KUKA KRL program: MyProgram_255().src

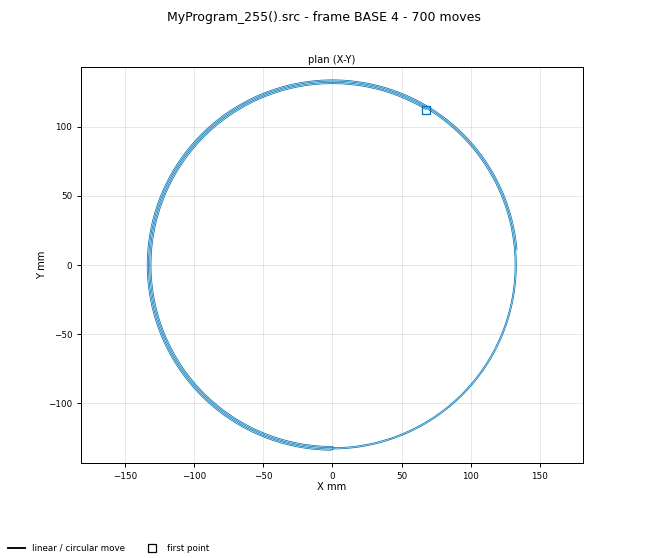
[picture p0: tool path of MyProgram_255().src in frame BASE 4, 700 of 700 moves have a stored position in this frame; points joined in program order, loops and branches not executed]
&ACCESS RVP
&REL 1
&PARAM TEMPLATE = C:\KRC\Roboter\Template\vorgabe
&PARAM EDITMASK = *
DEF MyProgram_255()
; ---- Setting reference (Base) ----
$BASE = BASE_DATA[4]

; --------------------------
; ---- Setting tool (TCP) ----
$TOOL = TOOL_DATA[3]
; --------------------------

$VEL.CP = VEL_APROX_PRINT
Startdeposition()
$VEL.CP = VEL_PRINT
LIN {X 67.662,Y 112.4887,Z 166,A 59.1873,B 11.341,C -0.0279,E1 11.4232,E2 391.3334} C_DIS
LIN {X 65.3064,Y 113.8724,Z 166,A 60.4715,B 11.341,C -0.0318,E1 11.4201,E2 390.0383} C_DIS
LIN {X 62.0567,Y 115.6751,Z 166,A 62.0322,B 11.341,C -0.0325,E1 11.4163,E2 388.4846} C_DIS
LIN {X 59.2043,Y 117.159,Z 166,A 63.3787,B 11.341,C -0.0329,E1 11.413,E2 387.1447} C_DIS
LIN {X 56.8476,Y 118.3202,Z 166,A 64.6326,B 11.341,C -0.037,E1 11.4098,E2 385.8781} C_DIS
LIN {X 53.382,Y 119.9236,Z 166,A 66.0531,B 11.341,C -0.0329,E1 11.4062,E2 384.4865} C_DIS
LIN {X 50.4227,Y 121.1975,Z 166,A 67.573,B 11.341,C -0.0372,E1 11.4023,E2 382.9533} C_DIS
LIN {X 47.4266,Y 122.401,Z 166,A 69.0048,B 11.341,C -0.0392,E1 11.3986,E2 381.519} C_DIS
LIN {X 44.4132,Y 123.5263,Z 166,A 70.3732,B 11.341,C -0.0397,E1 11.395,E2 380.1549} C_DIS
LIN {X 41.3721,Y 124.5778,Z 166,A 71.7718,B 11.341,C -0.0408,E1 11.3913,E2 378.7571} C_DIS
LIN {X 38.1151,Y 125.613,Z 166,A 73.257,B 11.341,C -0.0419,E1 11.3873,E2 377.2729} C_DIS
LIN {X 35.2196,Y 126.4551,Z 166,A 74.5585,B 11.341,C -0.0425,E1 11.3839,E2 375.9733} C_DIS
LIN {X 32.0679,Y 127.291,Z 166,A 75.9822,B 11.341,C -0.0435,E1 11.38,E2 374.5498} C_DIS
LIN {X 28.7806,Y 128.075,Z 166,A 77.4539,B 11.341,C -0.0443,E1 11.376,E2 373.0789} C_DIS
LIN {X 25.8073,Y 128.7068,Z 166,A 78.7946,B 11.341,C -0.0454,E1 11.3723,E2 371.7369} C_DIS
LIN {X 22.4469,Y 129.3365,Z 166,A 80.2607,B 11.341,C -0.0454,E1 11.3683,E2 370.2742} C_DIS
LIN {X 19.269,Y 129.8482,Z 166,A 81.6917,B 11.341,C -0.0466,E1 11.3644,E2 368.8407} C_DIS
LIN {X 16.0704,Y 130.2819,Z 166,A 83.0265,B 11.341,C -0.0453,E1 11.3607,E2 367.515} C_DIS
LIN {X 13.0675,Y 130.6173,Z 166,A 84.4622,B 11.341,C -0.0484,E1 11.3567,E2 366.0661} C_DIS
LIN {X 9.8613,Y 130.8977,Z 166,A 85.6593,B 11.341,C -0.0438,E1 11.3534,E2 364.8937} C_DIS
LIN {X 6.4486,Y 131.1099,Z 166,A 87.257,B 11.341,C -0.0464,E1 11.3489,E2 363.2843} C_DIS
LIN {X 3.2204,Y 131.2296,Z 166,A 88.6707,B 11.341,C -0.0466,E1 11.345,E2 361.8708} C_DIS
LIN {X 0.0025,Y 131.2704,Z 166,A 90.0792,B 11.341,C -0.0466,E1 11.341,E2 360.4626} C_DIS
LIN {X -3.2137,Y 131.2298,Z 166,A 91.4674,B 11.341,C -0.0461,E1 11.3372,E2 359.0768} C_DIS
LIN {X -6.4327,Y 131.1107,Z 166,A 92.8778,B 11.341,C -0.046,E1 11.3332,E2 357.6666} C_DIS
LIN {X -9.24,Y 130.9431,Z 166,A 94.2375,B 11.341,C -0.0487,E1 11.3294,E2 356.2921} C_DIS
LIN {X -12.6657,Y 130.6559,Z 166,A 95.6747,B 11.341,C -0.0468,E1 11.3254,E2 354.8631} C_DIS
LIN {X -16.0633,Y 130.2827,Z 166,A 97.1226,B 11.341,C -0.0452,E1 11.3214,E2 353.4212} C_DIS
LIN {X -19.0538,Y 129.8789,Z 166,A 98.4579,B 11.341,C -0.045,E1 11.3177,E2 352.0846} C_DIS
LIN {X -22.2446,Y 129.3713,Z 166,A 99.871,B 11.341,C -0.0443,E1 11.3138,E2 350.6721} C_DIS
LIN {X -25.4107,Y 128.7875,Z 166,A 101.3711,B 11.341,C -0.0456,E1 11.3097,E2 349.1619} C_DIS
LIN {X -28.5856,Y 128.1195,Z 166,A 102.7152,B 11.341,C -0.043,E1 11.306,E2 347.8271} C_DIS
LIN {X -31.9004,Y 127.3335,Z 166,A 104.1398,B 11.341,C -0.0405,E1 11.3022,E2 346.4108} C_DIS
LIN {X -34.8149,Y 126.5683,Z 166,A 105.5832,B 11.341,C -0.0423,E1 11.2983,E2 344.9533} C_DIS
LIN {X -37.9001,Y 125.6788,Z 166,A 106.9303,B 11.341,C -0.0398,E1 11.2947,E2 343.6137} C_DIS
LIN {X -41.1562,Y 124.6497,Z 166,A 108.4262,B 11.341,C -0.0385,E1 11.2907,E2 342.1182} C_DIS
LIN {X -44.2174,Y 123.5969,Z 166,A 109.8141,B 11.341,C -0.0365,E1 11.2871,E2 340.7344} C_DIS
LIN {X -47.0535,Y 122.546,Z 166,A 111.2316,B 11.341,C -0.0372,E1 11.2833,E2 339.3066} C_DIS
LIN {X -50.9887,Y 120.9611,Z 166,A 113.1889,B 11.341,C -0.0374,E1 11.2783,E2 337.3384} C_DIS
LIN {X -54.5865,Y 119.3812,Z 166,A 114.7862,B 11.341,C -0.0326,E1 11.2742,E2 335.7564} C_DIS
LIN {X -57.4016,Y 118.0545,Z 166,A 116.1867,B 11.341,C -0.0317,E1 11.2707,E2 334.3522} C_DIS
LIN {X -60.445,Y 116.5249,Z 166,A 117.565,B 11.341,C -0.0273,E1 11.2673,E2 332.9879} C_DIS
LIN {X -63.2703,Y 115.0164,Z 166,A 119.025,B 11.341,C -0.0266,E1 11.2637,E2 331.5219} C_DIS
LIN {X -66.0543,Y 113.4403,Z 166,A 120.4394,B 11.341,C -0.0249,E1 11.2603,E2 330.1066} C_DIS
LIN {X -68.7899,Y 111.8022,Z 166,A 121.854,B 11.341,C -0.0232,E1 11.2569,E2 328.6907} C_DIS
LIN {X -71.4124,Y 110.1455,Z 166,A 123.2027,B 11.341,C -0.0209,E1 11.2537,E2 327.3439} C_DIS
LIN {X -74.2646,Y 108.2429,Z 166,A 124.7098,B 11.341,C -0.0186,E1 11.2502,E2 325.837} C_DIS
LIN {X -76.7362,Y 106.5056,Z 166,A 126.0871,B 11.341,C -0.0175,E1 11.2471,E2 324.4541} C_DIS
LIN {X -79.4807,Y 104.4734,Z 166,A 127.6843,B 11.341,C -0.0171,E1 11.2435,E2 322.846} C_DIS
LIN {X -82.7236,Y 101.9251,Z 166,A 129.4945,B 11.341,C -0.0139,E1 11.2396,E2 321.0365} C_DIS
LIN {X -85.8192,Y 99.3321,Z 166,A 131.2791,B 11.341,C -0.0109,E1 11.2358,E2 319.2511} C_DIS
LIN {X -89.2655,Y 96.2471,Z 166,A 133.1947,B 11.341,C -0.0046,E1 11.2318,E2 317.3496} C_DIS
LIN {X -91.6701,Y 93.96,Z 166,A 134.657,B 11.341,C -0.0019,E1 11.2289,E2 315.8872} C_DIS
LIN {X -94.4472,Y 91.1675,Z 166,A 136.4062,B 11.341,C 0.0011,E1 11.2255,E2 314.1364} C_DIS
LIN {X -97.2631,Y 88.157,Z 166,A 138.3273,B 11.341,C 0.0026,E1 11.2218,E2 312.203} C_DIS
LIN {X -99.9831,Y 85.0597,Z 166,A 140.1409,B 11.341,C 0.0064,E1 11.2185,E2 310.3896} C_DIS
LIN {X -102.928,Y 81.4722,Z 166,A 142.0744,B 11.341,C 0.013,E1 11.2151,E2 308.4692} C_DIS
LIN {X -105.3163,Y 78.3596,Z 166,A 143.7874,B 11.341,C 0.0171,E1 11.2123,E2 306.758} C_DIS
LIN {X -107.3212,Y 75.5906,Z 166,A 145.2527,B 11.341,C 0.0212,E1 11.2099,E2 305.2975} C_DIS
LIN {X -109.0304,Y 73.104,Z 166,A 146.6964,B 11.341,C 0.0219,E1 11.2076,E2 303.8404} C_DIS
LIN {X -111.2462,Y 69.6864,Z 166,A 148.6229,B 11.341,C 0.0234,E1 11.2047,E2 301.8986} C_DIS
LIN {X -113.3192,Y 66.2616,Z 166,A 150.1978,B 11.341,C 0.0314,E1 11.2025,E2 300.3459} C_DIS
LIN {X -114.9075,Y 63.4669,Z 166,A 151.6157,B 11.341,C 0.0347,E1 11.2006,E2 298.9278} C_DIS
LIN {X -116.3051,Y 60.8637,Z 166,A 152.958,B 11.341,C 0.037,E1 11.1988,E2 297.5807} C_DIS
LIN {X -117.8767,Y 57.7619,Z 166,A 154.4808,B 11.341,C 0.041,E1 11.1969,E2 296.0591} C_DIS
LIN {X -119.2606,Y 54.8472,Z 166,A 155.8832,B 11.341,C 0.0449,E1 11.1952,E2 294.6589} C_DIS
LIN {X -120.5647,Y 51.9176,Z 166,A 157.2991,B 11.341,C 0.0483,E1 11.1937,E2 293.2427} C_DIS
LIN {X -121.7957,Y 48.9599,Z 166,A 158.7219,B 11.341,C 0.0517,E1 11.1922,E2 291.8187} C_DIS
LIN {X -123.0456,Y 45.7291,Z 166,A 160.2206,B 11.341,C 0.0562,E1 11.1907,E2 290.3232} C_DIS
LIN {X -124.0643,Y 42.8875,Z 166,A 161.581,B 11.341,C 0.059,E1 11.1894,E2 288.9594} C_DIS
LIN {X -125.0789,Y 39.8318,Z 166,A 163.141,B 11.3409,C 0.0598,E1 11.1881,E2 287.3828} C_DIS
LIN {X -126.4587,Y 35.2069,Z 166,A 165.1656,B 11.3409,C 0.0675,E1 11.1865,E2 285.3702} C_DIS
LIN {X -127.3329,Y 31.9028,Z 166,A 166.6254,B 11.3409,C 0.0724,E1 11.1855,E2 283.9159} C_DIS
LIN {X -128.0762,Y 28.7751,Z 166,A 167.9722,B 11.3408,C 0.0776,E1 11.1846,E2 282.5773} C_DIS
LIN {X -128.7073,Y 25.805,Z 166,A 169.4267,B 11.3408,C 0.0788,E1 11.1838,E2 281.1091} C_DIS
LIN {X -129.3345,Y 22.4582,Z 166,A 170.9103,B 11.3408,C 0.0832,E1 11.1831,E2 279.6275} C_DIS
LIN {X -129.8441,Y 19.2974,Z 166,A 172.3494,B 11.3408,C 0.0865,E1 11.1825,E2 278.185} C_DIS
LIN {X -130.2753,Y 16.1257,Z 166,A 173.682,B 11.3407,C 0.0919,E1 11.182,E2 276.8616} C_DIS
LIN {X -130.6063,Y 13.1817,Z 166,A 175.01,B 11.3407,C 0.0949,E1 11.1816,E2 275.5308} C_DIS
LIN {X -130.8983,Y 9.8531,Z 166,A 176.5923,B 11.3407,C 0.0967,E1 11.1812,E2 273.9355} C_DIS
LIN {X -131.1104,Y 6.4391,Z 166,A 177.9677,B 11.3406,C 0.1035,E1 11.181,E2 272.5755} C_DIS
LIN {X -131.2295,Y 3.2217,Z 166,A 179.447,B 11.3406,C 0.1061,E1 11.1809,E2 271.089} C_DIS
LIN {X -131.2723,Y 0.0074,Z 166,A -179.0626,B 11.3406,C 0.1085,E1 11.1809,E2 269.5899} C_DIS
LIN {X -131.1873,Y -4.6366,Z 166,A -176.9792,B 11.3405,C 0.1133,E1 11.181,E2 267.5019} C_DIS
LIN {X -131.0335,Y -7.8515,Z 166,A -175.6128,B 11.3405,C 0.1182,E1 11.1812,E2 266.1414} C_DIS
LIN {X -130.7845,Y -11.2613,Z 166,A -174.14,B 11.3404,C 0.123,E1 11.1815,E2 264.6724} C_DIS
LIN {X -130.4695,Y -14.4651,Z 166,A -172.7858,B 11.3404,C 0.1281,E1 11.1819,E2 263.3257} C_DIS
LIN {X -130.0967,Y -17.5042,Z 166,A -171.3374,B 11.3404,C 0.1297,E1 11.1824,E2 261.8653} C_DIS
LIN {X -129.6322,Y -20.6682,Z 166,A -169.9236,B 11.3403,C 0.1334,E1 11.183,E2 260.4508} C_DIS
LIN {X -129.0909,Y -23.8195,Z 166,A -168.5079,B 11.3403,C 0.137,E1 11.1837,E2 259.034} C_DIS
LIN {X -128.4298,Y -27.1555,Z 166,A -167.0467,B 11.3402,C 0.1417,E1 11.1845,E2 257.577} C_DIS
LIN {X -127.7642,Y -30.1336,Z 166,A -165.5785,B 11.3402,C 0.1428,E1 11.1855,E2 256.0938} C_DIS
LIN {X -126.9882,Y -33.2511,Z 166,A -164.222,B 11.3402,C 0.1477,E1 11.1864,E2 254.744} C_DIS
LIN {X -126.079,Y -36.5443,Z 166,A -162.78,B 11.34,C 0.1528,E1 11.1875,E2 253.309} C_DIS
LIN {X -125.199,Y -39.4556,Z 166,A -161.3122,B 11.34,C 0.1537,E1 11.1887,E2 251.8258} C_DIS
LIN {X -124.1294,Y -42.6997,Z 166,A -159.8592,B 11.34,C 0.1585,E1 11.19,E2 250.3785} C_DIS
LIN {X -123.0445,Y -45.732,Z 166,A -158.5033,B 11.3399,C 0.1634,E1 11.1913,E2 249.0297} C_DIS
LIN {X -121.8872,Y -48.7329,Z 166,A -157.0137,B 11.3399,C 0.1654,E1 11.1928,E2 247.531} C_DIS
LIN {X -120.3465,Y -52.4224,Z 166,A -155.212,B 11.3399,C 0.1689,E1 11.1948,E2 245.7239} C_DIS
LIN {X -118.6723,Y -56.1107,Z 166,A -153.5507,B 11.3397,C 0.1758,E1 11.1967,E2 244.0767} C_DIS
LIN {X -117.5193,Y -58.4864,Z 166,A -152.1926,B 11.3397,C 0.1745,E1 11.1984,E2 242.6951} C_DIS
LIN {X -115.6777,Y -62.0519,Z 166,A -150.4062,B 11.3397,C 0.1782,E1 11.2008,E2 240.9058} C_DIS
LIN {X -113.4207,Y -66.0882,Z 166,A -148.4733,B 11.3396,C 0.1851,E1 11.2034,E2 238.9844} C_DIS
LIN {X -111.7576,Y -68.8628,Z 166,A -147.0469,B 11.3396,C 0.1882,E1 11.2055,E2 237.5572} C_DIS
LIN {X -110.3098,Y -71.1593,Z 166,A -145.7766,B 11.3395,C 0.1893,E1 11.2074,E2 236.2774} C_DIS
LIN {X -108.241,Y -74.2674,Z 166,A -144.1303,B 11.3395,C 0.1928,E1 11.21,E2 234.6302} C_DIS
LIN {X -105.7565,Y -77.7645,Z 166,A -142.2177,B 11.3394,C 0.1963,E1 11.2131,E2 232.7138} C_DIS
LIN {X -103.4932,Y -80.7533,Z 166,A -140.5087,B 11.3394,C 0.1985,E1 11.2161,E2 230.9971} C_DIS
LIN {X -100.8567,Y -84.0229,Z 166,A -138.712,B 11.3393,C 0.2033,E1 11.2192,E2 229.2057} C_DIS
LIN {X -98.2956,Y -87.0043,Z 166,A -136.9297,B 11.3393,C 0.2055,E1 11.2225,E2 227.4161} C_DIS
LIN {X -95.6929,Y -89.8595,Z 166,A -135.327,B 11.3391,C 0.2108,E1 11.2256,E2 225.8243} C_DIS
LIN {X -92.8239,Y -92.8206,Z 166,A -133.4053,B 11.3391,C 0.2118,E1 11.2294,E2 223.8887} C_DIS
LIN {X -89.8627,Y -95.6898,Z 166,A -131.5943,B 11.3391,C 0.2151,E1 11.233,E2 222.0769} C_DIS
LIN {X -86.5059,Y -98.7347,Z 166,A -129.6375,B 11.339,C 0.2192,E1 11.2371,E2 220.1234} C_DIS
LIN {X -83.2718,Y -101.4773,Z 166,A -127.8857,B 11.3389,C 0.2247,E1 11.2408,E2 218.384} C_DIS
LIN {X -80.1684,Y -103.9465,Z 166,A -125.9969,B 11.3389,C 0.2242,E1 11.245,E2 216.4768} C_DIS
LIN {X -77.067,Y -106.2659,Z 166,A -124.4918,B 11.3387,C 0.2311,E1 11.2483,E2 214.9944} C_DIS
LIN {X -74.4424,Y -108.1209,Z 166,A -123.0232,B 11.3387,C 0.2318,E1 11.2517,E2 213.5181} C_DIS
LIN {X -72.1579,Y -109.6586,Z 166,A -121.6777,B 11.3387,C 0.2305,E1 11.2549,E2 212.1556} C_DIS
LIN {X -69.0408,Y -111.648,Z 166,A -120.1753,B 11.3387,C 0.2353,E1 11.2584,E2 210.6669} C_DIS
LIN {X -66.2691,Y -113.3148,Z 166,A -118.7593,B 11.3387,C 0.2372,E1 11.2618,E2 209.2505} C_DIS
LIN {X -63.9002,Y -114.6676,Z 166,A -117.4579,B 11.3387,C 0.2363,E1 11.265,E2 207.936} C_DIS
LIN {X -60.4624,Y -116.5158,Z 166,A -115.8994,B 11.3385,C 0.2417,E1 11.2688,E2 206.395} C_DIS
LIN {X -57.8004,Y -117.8577,Z 166,A -114.5216,B 11.3385,C 0.2415,E1 11.2723,E2 205.008} C_DIS
LIN {X -55.105,Y -119.1414,Z 166,A -113.1832,B 11.3385,C 0.2422,E1 11.2757,E2 203.6653} C_DIS
LIN {X -51.907,Y -120.5693,Z 166,A -111.6942,B 11.3385,C 0.2447,E1 11.2795,E2 202.1811} C_DIS
LIN {X -48.9276,Y -121.8087,Z 166,A -110.2816,B 11.3385,C 0.246,E1 11.2831,E2 200.7679} C_DIS
LIN {X -45.7401,Y -123.0415,Z 166,A -108.8104,B 11.3384,C 0.2479,E1 11.287,E2 199.2991} C_DIS
LIN {X -42.898,Y -124.0607,Z 166,A -107.4616,B 11.3384,C 0.2483,E1 11.2905,E2 197.9464} C_DIS
LIN {X -39.8469,Y -125.074,Z 166,A -106.0229,B 11.3384,C 0.2486,E1 11.2944,E2 196.5033} C_DIS
LIN {X -36.6683,Y -126.0428,Z 166,A -104.616,B 11.3384,C 0.2506,E1 11.2981,E2 195.1014} C_DIS
LIN {X -33.4679,Y -126.9304,Z 166,A -103.1835,B 11.3383,C 0.252,E1 11.302,E2 193.6707} C_DIS
LIN {X -30.5578,Y -127.6619,Z 166,A -101.8046,B 11.3383,C 0.2511,E1 11.3058,E2 192.2832} C_DIS
LIN {X -27.1923,Y -128.4218,Z 166,A -100.3413,B 11.3383,C 0.2529,E1 11.3097,E2 190.8247} C_DIS
LIN {X -24.3174,Y -128.9965,Z 166,A -99.0195,B 11.3383,C 0.2524,E1 11.3134,E2 189.4974} C_DIS
LIN {X -21.2035,Y -129.545,Z 166,A -97.62,B 11.3383,C 0.2524,E1 11.3172,E2 188.0951} C_DIS
LIN {X -17.6666,Y -130.0754,Z 166,A -96.082,B 11.3383,C 0.2535,E1 11.3215,E2 186.5595} C_DIS
LIN {X -14.6746,Y -130.447,Z 166,A -94.7613,B 11.3383,C 0.2536,E1 11.3251,E2 185.2377} C_DIS
LIN {X -11.2704,Y -130.7838,Z 166,A -93.3281,B 11.3383,C 0.2552,E1 11.3291,E2 183.8112} C_DIS
LIN {X -7.3216,Y -131.066,Z 166,A -91.3755,B 11.3383,C 0.25,E1 11.3346,E2 181.8308} C_DIS
LIN {X -3.2255,Y -131.2294,Z 166,A -89.7976,B 11.3383,C 0.255,E1 11.339,E2 180.2776} C_DIS
LIN {X -0.0098,Y -131.2704,Z 166,A -88.3914,B 11.3383,C 0.2548,E1 11.3429,E2 178.8705} C_DIS
LIN {X -0.0098,Y -131.2704,Z 166,A -88.3914,B 11.3383,C 0.2548,E1 11.3429,E2 178.8705} C_DIS
Enddeposition()
LIN {X 0.9627,Y -132.1793,Z 166,A -87.9974,B 11.3378,C 0.2622,E1 11.3437,E2 178.5145} C_DIS
Startdeposition()
$VEL.CP = VEL_PRINT
LIN {X -3.5481,Y -132.1372,Z 166,A -90.5843,B 11.3375,C 0.2775,E1 11.3362,E2 181.179} C_DIS
LIN {X -6.8903,Y -132.0053,Z 166,A -91.9427,B 11.3375,C 0.2753,E1 11.3325,E2 182.5269} C_DIS
LIN {X -10.7823,Y -131.7447,Z 166,A -93.783,B 11.3375,C 0.2787,E1 11.3273,E2 184.386} C_DIS
LIN {X -14.7745,Y -131.3579,Z 166,A -95.3648,B 11.3375,C 0.2747,E1 11.3229,E2 185.9496} C_DIS
LIN {X -17.6438,Y -131.0027,Z 166,A -96.5893,B 11.3375,C 0.2737,E1 11.3195,E2 187.171} C_DIS
LIN {X -20.5621,Y -130.576,Z 166,A -98.0041,B 11.3375,C 0.2765,E1 11.3156,E2 188.6027} C_DIS
LIN {X -25.0988,Y -129.7801,Z 166,A -100.0228,B 11.3375,C 0.2762,E1 11.31,E2 190.6245} C_DIS
LIN {X -28.9268,Y -128.9816,Z 166,A -101.6475,B 11.3375,C 0.2738,E1 11.3056,E2 192.2413} C_DIS
LIN {X -34.998,Y -127.4687,Z 166,A -104.2527,B 11.3376,C 0.2697,E1 11.2986,E2 194.8342} C_DIS
LIN {X -40.1602,Y -125.936,Z 166,A -106.718,B 11.3376,C 0.271,E1 11.292,E2 197.3157} C_DIS
LIN {X -43.9608,Y -124.6621,Z 166,A -108.3852,B 11.3376,C 0.268,E1 11.2876,E2 198.9747} C_DIS
LIN {X -48.0714,Y -123.1335,Z 166,A -110.3817,B 11.3376,C 0.2684,E1 11.2824,E2 200.9827} C_DIS
LIN {X -51.2743,Y -121.835,Z 166,A -111.8429,B 11.3377,C 0.266,E1 11.2786,E2 202.4396} C_DIS
LIN {X -55.0333,Y -120.1842,Z 166,A -113.6609,B 11.3377,C 0.265,E1 11.2739,E2 204.2621} C_DIS
LIN {X -59.3109,Y -118.1331,Z 166,A -115.6519,B 11.3378,C 0.2611,E1 11.269,E2 206.2454} C_DIS
LIN {X -62.9156,Y -116.254,Z 166,A -117.5195,B 11.3378,C 0.2612,E1 11.2643,E2 208.1255} C_DIS
LIN {X -66.402,Y -114.2979,Z 166,A -119.2831,B 11.3378,C 0.2596,E1 11.26,E2 209.8926} C_DIS
LIN {X -69.7189,Y -112.3054,Z 166,A -120.8703,B 11.338,C 0.2552,E1 11.2563,E2 211.4688} C_DIS
LIN {X -72.6717,Y -110.4175,Z 166,A -122.5068,B 11.338,C 0.2555,E1 11.2524,E2 213.1191} C_DIS
LIN {X -76.4072,Y -107.8666,Z 166,A -124.3738,B 11.338,C 0.2504,E1 11.2482,E2 214.9745} C_DIS
LIN {X -79.3283,Y -105.7372,Z 166,A -125.9122,B 11.3382,C 0.2472,E1 11.2447,E2 216.5091} C_DIS
LIN {X -81.708,Y -103.9086,Z 166,A -127.3283,B 11.3382,C 0.2475,E1 11.2416,E2 217.9386} C_DIS
LIN {X -86.5739,Y -99.8906,Z 166,A -130.0328,B 11.3382,C 0.2419,E1 11.2358,E2 220.6387} C_DIS
LIN {X -89.4536,Y -97.3204,Z 166,A -131.8115,B 11.3382,C 0.241,E1 11.2321,E2 222.4293} C_DIS
LIN {X -92.6327,Y -94.2994,Z 166,A -133.7286,B 11.3384,C 0.2376,E1 11.2282,E2 224.3476} C_DIS
LIN {X -95.7987,Y -91.082,Z 166,A -135.7454,B 11.3384,C 0.235,E1 11.2243,E2 226.3708} C_DIS
LIN {X -100.2187,Y -86.1938,Z 166,A -138.4156,B 11.3386,C 0.225,E1 11.2194,E2 229.0175} C_DIS
LIN {X -102.9955,Y -82.8561,Z 166,A -140.4726,B 11.3386,C 0.2245,E1 11.2157,E2 231.0944} C_DIS
LIN {X -105.3656,Y -79.8207,Z 166,A -142.1033,B 11.3387,C 0.2199,E1 11.2129,E2 232.7196} C_DIS
LIN {X -107.296,Y -77.2069,Z 166,A -143.6343,B 11.3387,C 0.2193,E1 11.2104,E2 234.2643} C_DIS
LIN {X -109.424,Y -74.1592,Z 166,A -145.2603,B 11.3387,C 0.2158,E1 11.2078,E2 235.8912} C_DIS
LIN {X -111.7157,Y -70.6599,Z 166,A -146.9595,B 11.3389,C 0.209,E1 11.2052,E2 237.5757} C_DIS
LIN {X -113.759,Y -67.3221,Z 166,A -148.8423,B 11.3389,C 0.2087,E1 11.2025,E2 239.4796} C_DIS
LIN {X -115.549,Y -64.2002,Z 166,A -150.2105,B 11.3391,C 0.2008,E1 11.2007,E2 240.824} C_DIS
LIN {X -117.4167,Y -60.7179,Z 166,A -152.0082,B 11.3391,C 0.1982,E1 11.1983,E2 242.6305} C_DIS
LIN {X -120.4535,Y -54.4416,Z 166,A -155.1893,B 11.3391,C 0.1936,E1 11.1945,E2 245.8282} C_DIS
LIN {X -121.9218,Y -51.0664,Z 166,A -156.7285,B 11.3393,C 0.1882,E1 11.1928,E2 247.3595} C_DIS
LIN {X -123.2326,Y -47.8165,Z 166,A -158.3019,B 11.3393,C 0.1852,E1 11.1912,E2 248.9381} C_DIS
LIN {X -124.4563,Y -44.5356,Z 166,A -159.7167,B 11.3394,C 0.179,E1 11.1898,E2 250.3395} C_DIS
LIN {X -125.4508,Y -41.6512,Z 166,A -161.1009,B 11.3394,C 0.1766,E1 11.1886,E2 251.7298} C_DIS
LIN {X -126.49,Y -38.381,Z 166,A -162.936,B 11.3394,C 0.1795,E1 11.187,E2 253.6047} C_DIS
LIN {X -127.439,Y -35.1039,Z 166,A -164.1022,B 11.3396,C 0.169,E1 11.1862,E2 254.7328} C_DIS
LIN {X -128.2028,Y -32.2005,Z 166,A -165.441,B 11.3396,C 0.1661,E1 11.1853,E2 256.0748} C_DIS
LIN {X -129.1394,Y -28.211,Z 166,A -167.9125,B 11.3395,C 0.175,E1 11.1837,E2 258.6261} C_DIS
LIN {X -130.1453,Y -23.1299,Z 166,A -169.4206,B 11.3398,C 0.1538,E1 11.183,E2 260.0458} C_DIS
LIN {X -131.0761,Y -17.0832,Z 166,A -172.1888,B 11.3398,C 0.1485,E1 11.1819,E2 262.8252} C_DIS
LIN {X -131.5276,Y -13.1748,Z 166,A -173.9683,B 11.3398,C 0.145,E1 11.1813,E2 264.6119} C_DIS
LIN {X -131.8436,Y -9.491,Z 166,A -175.6102,B 11.3399,C 0.1411,E1 11.181,E2 266.2567} C_DIS
LIN {X -132.0725,Y -5.4547,Z 166,A -177.3516,B 11.34,C 0.1357,E1 11.1807,E2 267.995} C_DIS
LIN {X -132.1683,Y -2.0896,Z 166,A -178.7968,B 11.34,C 0.1312,E1 11.1807,E2 269.4371} C_DIS
LIN {X -132.179,Y 1.437,Z 166,A 179.6148,B 11.3401,C 0.1279,E1 11.1807,E2 271.0309} C_DIS
LIN {X -132.0879,Y 5.0617,Z 166,A 178.0274,B 11.3401,C 0.1236,E1 11.1807,E2 272.6185} C_DIS
LIN {X -131.8611,Y 9.2516,Z 166,A 176.1759,B 11.3401,C 0.1189,E1 11.1811,E2 274.4719} C_DIS
LIN {X -131.5553,Y 12.8864,Z 166,A 174.6147,B 11.3403,C 0.1138,E1 11.1815,E2 276.029} C_DIS
LIN {X -130.7873,Y 19.1749,Z 166,A 171.5775,B 11.3403,C 0.1116,E1 11.1826,E2 279.0973} C_DIS
LIN {X -130.0788,Y 23.5011,Z 166,A 169.9122,B 11.3403,C 0.1014,E1 11.1834,E2 280.733} C_DIS
LIN {X -129.4416,Y 26.7919,Z 166,A 168.0038,B 11.3403,C 0.1063,E1 11.1845,E2 282.693} C_DIS
LIN {X -128.6,Y 30.5768,Z 166,A 166.6692,B 11.3404,C 0.0945,E1 11.1853,E2 283.9854} C_DIS
LIN {X -127.7264,Y 34.0396,Z 166,A 165.1741,B 11.3404,C 0.089,E1 11.1863,E2 285.4725} C_DIS
LIN {X -126.6616,Y 37.816,Z 166,A 163.4553,B 11.3405,C 0.0846,E1 11.1877,E2 287.1916} C_DIS
LIN {X -125.808,Y 40.561,Z 166,A 162.1921,B 11.3405,C 0.0814,E1 11.1887,E2 288.4554} C_DIS
LIN {X -124.8755,Y 43.3452,Z 166,A 160.8136,B 11.3405,C 0.0799,E1 11.19,E2 289.8448} C_DIS
LIN {X -123.7018,Y 46.5898,Z 166,A 159.3856,B 11.3405,C 0.0744,E1 11.1914,E2 291.2632} C_DIS
LIN {X -122.4123,Y 49.8815,Z 166,A 157.3407,B 11.3405,C 0.0804,E1 11.1936,E2 293.366} C_DIS
LIN {X -120.8023,Y 53.6618,Z 166,A 155.9611,B 11.3406,C 0.0676,E1 11.1951,E2 294.6969} C_DIS
LIN {X -118.8847,Y 57.7887,Z 166,A 154.0809,B 11.3406,C 0.0604,E1 11.1973,E2 296.5641} C_DIS
LIN {X -117.7882,Y 59.9884,Z 166,A 152.857,B 11.3406,C 0.0607,E1 11.1988,E2 297.8052} C_DIS
LIN {X -116.0492,Y 63.2912,Z 166,A 151.3783,B 11.3406,C 0.0537,E1 11.2008,E2 299.2659} C_DIS
LIN {X -114.2437,Y 66.4951,Z 166,A 149.7474,B 11.3407,C 0.0503,E1 11.203,E2 300.8994} C_DIS
LIN {X -111.878,Y 70.4027,Z 166,A 147.4577,B 11.3407,C 0.0516,E1 11.2064,E2 303.2228} C_DIS
LIN {X -109.2257,Y 74.4521,Z 166,A 145.444,B 11.3407,C 0.0447,E1 11.2095,E2 305.2244} C_DIS
LIN {X -106.7687,Y 77.9346,Z 166,A 143.566,B 11.3407,C 0.0408,E1 11.2126,E2 307.1039} C_DIS
LIN {X -104.2939,Y 81.2162,Z 166,A 141.7827,B 11.3407,C 0.0366,E1 11.2156,E2 308.8854} C_DIS
LIN {X -101.483,Y 84.7025,Z 166,A 139.8758,B 11.3407,C 0.0314,E1 11.219,E2 310.7862} C_DIS
LIN {X -98.7041,Y 87.9251,Z 166,A 138.036,B 11.3407,C 0.0271,E1 11.2224,E2 312.6235} C_DIS
LIN {X -95.9035,Y 90.9717,Z 166,A 136.2133,B 11.3407,C 0.0238,E1 11.2258,E2 314.4475} C_DIS
LIN {X -93.2084,Y 93.7304,Z 166,A 134.4678,B 11.3407,C 0.0218,E1 11.2293,E2 316.1998} C_DIS
LIN {X -90.1698,Y 96.6572,Z 166,A 132.6495,B 11.3408,C 0.0178,E1 11.233,E2 318.015} C_DIS
LIN {X -87.147,Y 99.3916,Z 166,A 130.8111,B 11.3408,C 0.0157,E1 11.2368,E2 319.8599} C_DIS
LIN {X -83.671,Y 102.3345,Z 166,A 128.852,B 11.3408,C 0.0116,E1 11.241,E2 321.8152} C_DIS
LIN {X -80.4137,Y 104.9135,Z 166,A 127.0637,B 11.3408,C 0.008,E1 11.2449,E2 323.6003} C_DIS
LIN {X -77.3577,Y 107.187,Z 166,A 125.3784,B 11.3408,C 0.0058,E1 11.2487,E2 325.2879} C_DIS
LIN {X -73.6429,Y 109.7726,Z 166,A 123.3812,B 11.3408,C 0.0032,E1 11.2534,E2 327.2873} C_DIS
LIN {X -69.84,Y 112.23,Z 166,A 121.4918,B 11.3408,C -0.0016,E1 11.2578,E2 329.1664} C_DIS
LIN {X -64.4414,Y 115.4151,Z 166,A 118.6279,B 11.3408,C -0.0026,E1 11.2647,E2 332.0448} C_DIS
LIN {X -61.1977,Y 117.1648,Z 166,A 117.1535,B 11.3408,C -0.0075,E1 11.2683,E2 333.5035} C_DIS
LIN {X -58.2534,Y 118.6561,Z 166,A 115.724,B 11.3408,C -0.0095,E1 11.2719,E2 334.9315} C_DIS
LIN {X -52.6518,Y 121.2457,Z 166,A 112.9525,B 11.3408,C -0.0108,E1 11.279,E2 337.712} C_DIS
LIN {X -48.9305,Y 122.7956,Z 166,A 111.2223,B 11.3408,C -0.0132,E1 11.2834,E2 339.4388} C_DIS
LIN {X -44.7986,Y 124.3615,Z 166,A 109.2791,B 11.3408,C -0.0146,E1 11.2885,E2 341.3837} C_DIS
LIN {X -38.9801,Y 126.3066,Z 166,A 106.8985,B 11.3408,C -0.0233,E1 11.2948,E2 343.7299} C_DIS
LIN {X -34.8285,Y 127.516,Z 166,A 104.694,B 11.3408,C -0.0176,E1 11.3008,E2 345.9716} C_DIS
LIN {X -31.0574,Y 128.4842,Z 166,A 103.161,B 11.3408,C -0.0223,E1 11.3049,E2 347.4854} C_DIS
LIN {X -25.7992,Y 129.6436,Z 166,A 100.7895,B 11.3408,C -0.023,E1 11.3114,E2 349.8597} C_DIS
LIN {X -21.9761,Y 130.3452,Z 166,A 99.0916,B 11.3408,C -0.0237,E1 11.316,E2 351.558} C_DIS
LIN {X -18.6805,Y 130.858,Z 166,A 97.6643,B 11.3408,C -0.0248,E1 11.32,E2 352.9823} C_DIS
LIN {X -15.4361,Y 131.2804,Z 166,A 96.1226,B 11.3408,C -0.0226,E1 11.3243,E2 354.5375} C_DIS
LIN {X -10.9024,Y 131.7345,Z 166,A 94.1987,B 11.3408,C -0.0244,E1 11.3296,E2 356.4544} C_DIS
LIN {X -7.1231,Y 131.9936,Z 166,A 92.5139,B 11.3408,C -0.0238,E1 11.3343,E2 358.1434} C_DIS
LIN {X -3.5616,Y 132.1369,Z 166,A 90.9488,B 11.3408,C -0.0236,E1 11.3387,E2 359.7099} C_DIS
LIN {X 0.1908,Y 132.1858,Z 166,A 89.3327,B 11.3408,C -0.024,E1 11.3432,E2 361.3242} C_DIS
LIN {X 3.9208,Y 132.1269,Z 166,A 87.8581,B 11.3408,C -0.0272,E1 11.3473,E2 362.7814} C_DIS
LIN {X 7.3388,Y 131.9826,Z 166,A 86.3652,B 11.3408,C -0.0268,E1 11.3514,E2 364.275} C_DIS
LIN {X 11.482,Y 131.6856,Z 166,A 84.5479,B 11.3408,C -0.0261,E1 11.3565,E2 366.0934} C_DIS
LIN {X 14.2529,Y 131.414,Z 166,A 83.352,B 11.3408,C -0.0261,E1 11.3598,E2 367.2877} C_DIS
LIN {X 17.3054,Y 131.047,Z 166,A 81.9399,B 11.3408,C -0.0238,E1 11.3637,E2 368.7085} C_DIS
LIN {X 21.6847,Y 130.3938,Z 166,A 79.9789,B 11.3408,C -0.0221,E1 11.3692,E2 370.6739} C_DIS
LIN {X 25.7769,Y 129.6482,Z 166,A 78.1988,B 11.3408,C -0.0217,E1 11.374,E2 372.4509} C_DIS
LIN {X 31.3948,Y 128.4028,Z 166,A 75.7743,B 11.3408,C -0.0218,E1 11.3806,E2 374.8667} C_DIS
LIN {X 37.3211,Y 126.8065,Z 166,A 73.0355,B 11.3408,C -0.018,E1 11.388,E2 377.6142} C_DIS
LIN {X 40.7946,Y 125.7333,Z 166,A 71.5528,B 11.3408,C -0.0189,E1 11.3919,E2 379.0859} C_DIS
LIN {X 44.6681,Y 124.4086,Z 166,A 69.718,B 11.3408,C -0.0159,E1 11.3968,E2 380.9275} C_DIS
LIN {X 48.2829,Y 123.0513,Z 166,A 68.121,B 11.3408,C -0.016,E1 11.4009,E2 382.5155} C_DIS
LIN {X 52.1574,Y 121.4594,Z 166,A 66.3341,B 11.3408,C -0.0148,E1 11.4055,E2 384.299} C_DIS
LIN {X 55.5916,Y 119.9261,Z 166,A 64.6916,B 11.3408,C -0.0126,E1 11.4097,E2 385.9429} C_DIS
LIN {X 58.8648,Y 118.3545,Z 166,A 63.138,B 11.3408,C -0.0111,E1 11.4136,E2 387.4942} C_DIS
LIN {X 62.0016,Y 116.7427,Z 166,A 61.6458,B 11.3408,C -0.01,E1 11.4173,E2 388.9822} C_DIS
LIN {X 64.903,Y 115.1556,Z 166,A 60.0227,B 11.3408,C -0.0034,E1 11.4213,E2 390.6277} C_DIS
LIN {X 68.0801,Y 113.3069,Z 166,A 58.592,B 11.3408,C -0.005,E1 11.4247,E2 392.0397} C_DIS
LIN {X 71.4574,Y 111.2074,Z 166,A 56.7287,B 11.3408,C 0.001,E1 11.4291,E2 393.9196} C_DIS
LIN {X 75.1479,Y 108.7481,Z 166,A 54.8646,B 11.3408,C 0.0027,E1 11.4334,E2 395.7772} C_DIS
LIN {X 78.5579,Y 106.3108,Z 166,A 53.1359,B 11.3408,C 0.0035,E1 11.4373,E2 397.496} C_DIS
LIN {X 81.7351,Y 103.8873,Z 166,A 51.2943,B 11.3408,C 0.0093,E1 11.4414,E2 399.3509} C_DIS
LIN {X 84.2875,Y 101.8274,Z 166,A 49.9707,B 11.3408,C 0.0095,E1 11.4442,E2 400.6634} C_DIS
LIN {X 87.7168,Y 98.8888,Z 166,A 48.0574,B 11.3408,C 0.012,E1 11.4483,E2 402.5722} C_DIS
LIN {X 90.7514,Y 96.1113,Z 166,A 46.2601,B 11.3408,C 0.0159,E1 11.4519,E2 404.3718} C_DIS
LIN {X 93.6236,Y 93.3159,Z 166,A 44.5122,B 11.3408,C 0.0197,E1 11.4554,E2 406.1217} C_DIS
LIN {X 96.6964,Y 90.1277,Z 166,A 42.6164,B 11.3408,C 0.0231,E1 11.459,E2 408.0156} C_DIS
LIN {X 99.8334,Y 86.6407,Z 166,A 40.6337,B 11.3408,C 0.0262,E1 11.4627,E2 409.9933} C_DIS
LIN {X 103.3191,Y 82.4523,Z 166,A 38.2826,B 11.3408,C 0.0312,E1 11.4669,E2 412.3443} C_DIS
LIN {X 106.0108,Y 78.9614,Z 166,A 36.455,B 11.3408,C 0.0335,E1 11.4699,E2 414.1631} C_DIS
LIN {X 108.3485,Y 75.7223,Z 166,A 34.898,B 11.3408,C 0.033,E1 11.4724,E2 415.7005} C_DIS
LIN {X 109.7492,Y 73.6779,Z 166,A 33.7322,B 11.3408,C 0.038,E1 11.4743,E2 416.8778} C_DIS
LIN {X 111.5595,Y 70.9074,Z 166,A 32.1997,B 11.3408,C 0.044,E1 11.4766,E2 418.4228} C_DIS
LIN {X 114.3985,Y 66.2282,Z 166,A 30.107,B 11.3408,C 0.0427,E1 11.4796,E2 420.484} C_DIS
LIN {X 115.6749,Y 63.9728,Z 166,A 28.8023,B 11.3408,C 0.0502,E1 11.4814,E2 421.8109} C_DIS
LIN {X 117.4945,Y 60.5653,Z 166,A 26.9343,B 11.3407,C 0.0596,E1 11.4838,E2 423.703} C_DIS
LIN {X 119.592,Y 56.3115,Z 166,A 24.9848,B 11.3407,C 0.0622,E1 11.4862,E2 425.6415} C_DIS
LIN {X 121.3091,Y 52.5051,Z 166,A 23.3016,B 11.3407,C 0.0637,E1 11.4881,E2 427.3109} C_DIS
LIN {X 122.8718,Y 48.7417,Z 166,A 21.635,B 11.3407,C 0.0659,E1 11.4898,E2 428.9673} C_DIS
LIN {X 124.117,Y 45.4767,Z 166,A 20.1749,B 11.3407,C 0.0686,E1 11.4912,E2 430.4221} C_DIS
LIN {X 124.9594,Y 43.1034,Z 166,A 18.9844,B 11.3406,C 0.0741,E1 11.4923,E2 431.6251} C_DIS
LIN {X 126.0736,Y 39.7293,Z 166,A 17.4316,B 11.3406,C 0.0788,E1 11.4937,E2 433.1809} C_DIS
LIN {X 127.0794,Y 36.387,Z 166,A 15.9293,B 11.3406,C 0.0827,E1 11.4949,E2 434.6831} C_DIS
LIN {X 128.3596,Y 31.5742,Z 166,A 13.8012,B 11.3405,C 0.088,E1 11.4963,E2 436.8095} C_DIS
LIN {X 129.2165,Y 27.8538,Z 166,A 12.2557,B 11.3405,C 0.0899,E1 11.4973,E2 438.3436} C_DIS
LIN {X 129.9463,Y 24.2298,Z 166,A 10.6925,B 11.3405,C 0.0934,E1 11.4981,E2 439.9036} C_DIS
LIN {X 130.6123,Y 20.3276,Z 166,A 8.9698,B 11.3404,C 0.0986,E1 11.4989,E2 441.6287} C_DIS
LIN {X 131.106,Y 16.8548,Z 166,A 7.3603,B 11.3404,C 0.1054,E1 11.4995,E2 443.2503} C_DIS
LIN {X 131.5837,Y 12.5906,Z 166,A 5.6027,B 11.3404,C 0.1081,E1 11.5,E2 444.9976} C_DIS
LIN {X 131.9037,Y 8.6299,Z 166,A 3.8912,B 11.3403,C 0.1128,E1 11.5003,E2 446.7096} C_DIS
LIN {X 132.089,Y 5.0313,Z 166,A 2.4064,B 11.3403,C 0.1154,E1 11.5005,E2 448.1867} C_DIS
LIN {X 132.1809,Y 1.1603,Z 166,A 0.811,B 11.3403,C 0.1181,E1 11.5006,E2 449.7739} C_DIS
LIN {X 132.1666,Y -2.1972,Z 166,A -0.7243,B 11.3401,C 0.1245,E1 11.5006,E2 451.3203} C_DIS
LIN {X 132.0287,Y -6.4256,Z 166,A -2.5224,B 11.3401,C 0.129,E1 11.5004,E2 453.1161} C_DIS
LIN {X 131.803,Y -10.0466,Z 166,A -4.0423,B 11.3401,C 0.1322,E1 11.5001,E2 454.6314} C_DIS
LIN {X 131.5353,Y -13.0944,Z 166,A -5.3126,B 11.3401,C 0.1346,E1 11.4998,E2 455.8964} C_DIS
LIN {X 131.2109,Y -16.0188,Z 166,A -6.6099,B 11.34,C 0.139,E1 11.4993,E2 457.1977} C_DIS
LIN {X 130.6667,Y -19.976,Z 166,A -8.3004,B 11.34,C 0.1429,E1 11.4987,E2 458.8853} C_DIS
LIN {X 130.083,Y -23.4777,Z 166,A -9.8787,B 11.3399,C 0.1485,E1 11.4979,E2 460.4699} C_DIS
LIN {X 129.3554,Y -27.2107,Z 166,A -12.109,B 11.3396,C 0.1687,E1 11.4966,E2 462.7716} C_DIS
LIN {X 128.2416,Y -32.0478,Z 166,A -13.4592,B 11.3398,C 0.1537,E1 11.4958,E2 464.0285} C_DIS
LIN {X 127.0755,Y -36.4023,Z 166,A -15.5121,B 11.3397,C 0.1619,E1 11.4943,E2 466.0956} C_DIS
LIN {X 126.0127,Y -39.9201,Z 166,A -17.2474,B 11.3396,C 0.1702,E1 11.4928,E2 467.8497} C_DIS
LIN {X 124.8057,Y -43.5466,Z 166,A -18.8197,B 11.3396,C 0.1727,E1 11.4914,E2 469.4138} C_DIS
LIN {X 123.1785,Y -47.9557,Z 166,A -20.7476,B 11.3395,C 0.1755,E1 11.4895,E2 471.3309} C_DIS
LIN {X 121.8948,Y -51.1311,Z 166,A -22.2646,B 11.3394,C 0.1804,E1 11.4879,E2 472.8535} C_DIS
LIN {X 120.3524,Y -54.6678,Z 166,A -25.1269,B 11.3388,C 0.2162,E1 11.4844,E2 475.8594} C_DIS
LIN {X 116.6915,Y -62.0991,Z 166,A -27.9035,B 11.339,C 0.2045,E1 11.4809,E2 478.5437} C_DIS
LIN {X 114.6093,Y -65.8641,Z 166,A -29.2529,B 11.3391,C 0.1959,E1 11.4791,E2 479.8335} C_DIS
LIN {X 112.5775,Y -69.2786,Z 166,A -30.918,B 11.3391,C 0.1988,E1 11.4767,E2 481.4936} C_DIS
LIN {X 110.8795,Y -71.9648,Z 166,A -32.4089,B 11.339,C 0.2053,E1 11.4745,E2 482.9998} C_DIS
LIN {X 108.3155,Y -75.7697,Z 166,A -34.4093,B 11.3389,C 0.2106,E1 11.4713,E2 485.0037} C_DIS
LIN {X 105.7174,Y -79.3545,Z 166,A -36.3143,B 11.3389,C 0.2149,E1 11.4681,E2 486.9092} C_DIS
LIN {X 102.8405,Y -83.0483,Z 166,A -38.4527,B 11.3387,C 0.2226,E1 11.4644,E2 489.063} C_DIS
LIN {X 100.4393,Y -85.9379,Z 166,A -39.9266,B 11.3387,C 0.2223,E1 11.4618,E2 490.5202} C_DIS
LIN {X 97.4774,Y -89.2827,Z 166,A -41.7418,B 11.3387,C 0.2236,E1 11.4584,E2 492.3229} C_DIS
LIN {X 94.9714,Y -91.9436,Z 166,A -43.4125,B 11.3385,C 0.2293,E1 11.4552,E2 494.0057} C_DIS
LIN {X 91.7664,Y -95.143,Z 166,A -45.3124,B 11.3385,C 0.2319,E1 11.4514,E2 495.9001} C_DIS
LIN {X 88.973,Y -97.7601,Z 166,A -46.9798,B 11.3384,C 0.2356,E1 11.448,E2 497.5703} C_DIS
LIN {X 85.5432,Y -100.7748,Z 166,A -48.9725,B 11.3384,C 0.2399,E1 11.4437,E2 499.5666} C_DIS
LIN {X 82.54,Y -103.2493,Z 166,A -50.5289,B 11.3384,C 0.2399,E1 11.4404,E2 501.109} C_DIS
LIN {X 79.6998,Y -105.4568,Z 166,A -52.0576,B 11.3383,C 0.242,E1 11.437,E2 502.6356} C_DIS
LIN {X 77.2018,Y -107.2997,Z 166,A -53.5225,B 11.3381,C 0.2476,E1 11.4337,E2 504.1164} C_DIS
LIN {X 73.5506,Y -109.8341,Z 166,A -55.5192,B 11.3381,C 0.2527,E1 11.429,E2 506.1234} C_DIS
LIN {X 69.9632,Y -112.1533,Z 166,A -57.2313,B 11.3381,C 0.2523,E1 11.425,E2 507.8204} C_DIS
LIN {X 66.5872,Y -114.1907,Z 166,A -58.8909,B 11.3381,C 0.2538,E1 11.4211,E2 509.4758} C_DIS
LIN {X 63.0428,Y -116.1847,Z 166,A -60.7469,B 11.3379,C 0.2589,E1 11.4165,E2 511.3446} C_DIS
LIN {X 59.3762,Y -118.0998,Z 166,A -62.3554,B 11.3379,C 0.2568,E1 11.4125,E2 512.9324} C_DIS
LIN {X 56.7675,Y -119.3741,Z 166,A -63.6195,B 11.3379,C 0.2587,E1 11.4094,E2 514.1983} C_DIS
LIN {X 53.9477,Y -120.6744,Z 166,A -64.9793,B 11.3379,C 0.2609,E1 11.4059,E2 515.5609} C_DIS
LIN {X 50.4453,Y -122.1812,Z 166,A -66.5654,B 11.3379,C 0.2613,E1 11.4018,E2 517.1405} C_DIS
LIN {X 47.0458,Y -123.531,Z 166,A -68.1303,B 11.3379,C 0.2627,E1 11.3978,E2 518.7042} C_DIS
LIN {X 44.1282,Y -124.6032,Z 166,A -69.8337,B 11.3376,C 0.273,E1 11.3932,E2 520.4516} C_DIS
LIN {X 40.9548,Y -125.6822,Z 166,A -70.9324,B 11.3377,C 0.2658,E1 11.3904,E2 521.5087} C_DIS
LIN {X 33.0839,Y -127.9786,Z 166,A -74.4959,B 11.3377,C 0.2694,E1 11.3808,E2 525.0761} C_DIS
LIN {X 30.2855,Y -128.6702,Z 166,A -75.9245,B 11.3375,C 0.2748,E1 11.3768,E2 526.5273} C_DIS
LIN {X 26.4865,Y -129.5038,Z 166,A -77.4272,B 11.3376,C 0.2715,E1 11.3728,E2 528.0089} C_DIS
LIN {X 22.6499,Y -130.2312,Z 166,A -79.0815,B 11.3376,C 0.2717,E1 11.3683,E2 529.6598} C_DIS
LIN {X 19.9028,Y -130.678,Z 166,A -80.3069,B 11.3376,C 0.2729,E1 11.3649,E2 530.8882} C_DIS
LIN {X 15.9178,Y -131.223,Z 166,A -82.1081,B 11.3376,C 0.2752,E1 11.3599,E2 532.6975} C_DIS
LIN {X 12.2971,Y -131.6119,Z 166,A -83.5528,B 11.3376,C 0.2726,E1 11.3559,E2 534.1269} C_DIS
LIN {X 8.9457,Y -131.8834,Z 166,A -85.2392,B 11.3374,C 0.2787,E1 11.3511,E2 535.8418} C_DIS
LIN {X 4.7739,Y -132.0991,Z 166,A -87.0037,B 11.3374,C 0.278,E1 11.3462,E2 537.6017} C_DIS
LIN {X 0.9627,Y -132.1793,Z 166,A -87.9958,B 11.3378,C 0.2625,E1 11.3437,E2 538.5145} C_DIS
Enddeposition()
LIN {X 0.9627,Y -132.1793,Z 166,A -87.9958,B 11.3378,C 0.2625,E1 11.3437,E2 538.5145} C_DIS
Startdeposition()
$VEL.CP = VEL_PRINT
LIN {X 1.6006,Y -133.093,Z 166,A -87.4623,B 11.3376,C 0.263,E1 11.345,E2 537.9838} C_DIS
LIN {X 5.8752,Y -132.9732,Z 166,A -85.6166,B 11.3376,C 0.2625,E1 11.3501,E2 536.1366} C_DIS
LIN {X 9.6604,Y -132.7501,Z 166,A -84.0983,B 11.3376,C 0.2647,E1 11.3543,E2 534.6314} C_DIS
LIN {X 13.7545,Y -132.3894,Z 166,A -82.3127,B 11.3376,C 0.2636,E1 11.3593,E2 532.8428} C_DIS
LIN {X 17.335,Y -131.9674,Z 166,A -80.7829,B 11.3376,C 0.2634,E1 11.3635,E2 531.3147} C_DIS
LIN {X 21.1406,Y -131.4137,Z 166,A -78.9869,B 11.3377,C 0.2589,E1 11.3685,E2 529.5005} C_DIS
LIN {X 24.9411,Y -130.7433,Z 166,A -77.5016,B 11.3377,C 0.2622,E1 11.3725,E2 528.0357} C_DIS
LIN {X 27.8456,Y -130.1558,Z 166,A -76.1901,B 11.3377,C 0.2604,E1 11.3761,E2 526.7189} C_DIS
LIN {X 32.0496,Y -129.1866,Z 166,A -73.6619,B 11.3381,C 0.2419,E1 11.3832,E2 524.1061} C_DIS
LIN {X 37.2295,Y -127.7882,Z 166,A -72.0253,B 11.3378,C 0.2568,E1 11.3874,E2 522.5514} C_DIS
LIN {X 44.175,Y -125.5578,Z 166,A -68.9626,B 11.3378,C 0.2555,E1 11.3955,E2 519.496} C_DIS
LIN {X 47.4817,Y -124.346,Z 166,A -67.4441,B 11.3378,C 0.2537,E1 11.3995,E2 517.9759} C_DIS
LIN {X 50.4857,Y -123.1568,Z 166,A -65.9525,B 11.3379,C 0.2494,E1 11.4034,E2 516.4708} C_DIS
LIN {X 54.1533,Y -121.5864,Z 166,A -64.3267,B 11.3379,C 0.2495,E1 11.4075,E2 514.8547} C_DIS
LIN {X 57.2062,Y -120.1802,Z 166,A -62.9342,B 11.3379,C 0.2489,E1 11.411,E2 513.4676} C_DIS
LIN {X 60.0301,Y -118.7953,Z 166,A -61.5284,B 11.338,C 0.2457,E1 11.4145,E2 512.0542} C_DIS
LIN {X 63.0442,Y -117.2252,Z 166,A -60.0441,B 11.338,C 0.2429,E1 11.4182,E2 510.566} C_DIS
LIN {X 66.9034,Y -115.0665,Z 166,A -58.1327,B 11.3381,C 0.2397,E1 11.4229,E2 508.6518} C_DIS
LIN {X 70.651,Y -112.8047,Z 166,A -55.7787,B 11.3384,C 0.2244,E1 11.4286,E2 506.2377} C_DIS
LIN {X 74.5977,Y -110.2338,Z 166,A -54.3149,B 11.3382,C 0.2356,E1 11.4318,E2 504.8419} C_DIS
LIN {X 77.7885,Y -108.0065,Z 166,A -52.5613,B 11.3383,C 0.2305,E1 11.4358,E2 503.077} C_DIS
LIN {X 81.2603,Y -105.4191,Z 166,A -50.6038,B 11.3384,C 0.2245,E1 11.4402,E2 501.106} C_DIS
LIN {X 86.5654,Y -101.1083,Z 166,A -47.787,B 11.3384,C 0.222,E1 11.4462,E2 498.3017} C_DIS
LIN {X 89.966,Y -98.094,Z 166,A -45.9833,B 11.3384,C 0.222,E1 11.4499,E2 496.5148} C_DIS
LIN {X 93.1944,Y -95.0322,Z 166,A -43.6592,B 11.3388,C 0.2071,E1 11.4547,E2 494.138} C_DIS
LIN {X 95.9845,Y -92.2139,Z 166,A -42.2598,B 11.3387,C 0.2115,E1 11.4574,E2 492.775} C_DIS
LIN {X 99.1298,Y -88.8234,Z 166,A -40.5543,B 11.3387,C 0.2146,E1 11.4605,E2 491.1025} C_DIS
LIN {X 100.899,Y -86.8085,Z 166,A -38.8882,B 11.3389,C 0.1983,E1 11.4637,E2 489.3719} C_DIS
LIN {X 103.3422,Y -83.886,Z 166,A -37.5319,B 11.3389,C 0.202,E1 11.466,E2 488.0488} C_DIS
LIN {X 105.7767,Y -80.7936,Z 166,A -35.9241,B 11.3389,C 0.2003,E1 11.4687,E2 486.4497} C_DIS
LIN {X 108.3916,Y -77.2503,Z 166,A -34.0353,B 11.3389,C 0.1958,E1 11.4718,E2 484.5597} C_DIS
LIN {X 110.9102,Y -73.5892,Z 166,A -32.2007,B 11.339,C 0.1931,E1 11.4747,E2 482.7325} C_DIS
LIN {X 113.0998,Y -70.1767,Z 166,A -30.4054,B 11.3391,C 0.1873,E1 11.4774,E2 480.929} C_DIS
LIN {X 115.0031,Y -67.013,Z 166,A -28.9738,B 11.3391,C 0.1874,E1 11.4794,E2 479.5151} C_DIS
LIN {X 116.8416,Y -63.7523,Z 166,A -27.2673,B 11.3392,C 0.1806,E1 11.4817,E2 477.795} C_DIS
LIN {X 118.4403,Y -60.7274,Z 166,A -25.4192,B 11.3394,C 0.1665,E1 11.4842,E2 475.8988} C_DIS
LIN {X 120.2364,Y -57.0879,Z 166,A -23.97,B 11.3394,C 0.1699,E1 11.4859,E2 474.4844} C_DIS
LIN {X 122.1477,Y -52.8748,Z 166,A -22.3453,B 11.3394,C 0.1743,E1 11.4876,E2 472.9026} C_DIS
LIN {X 123.3453,Y -50.0181,Z 166,A -20.8599,B 11.3394,C 0.1665,E1 11.4893,E2 471.3969} C_DIS
LIN {X 124.8618,Y -46.1055,Z 166,A -18.9859,B 11.3395,C 0.1597,E1 11.4911,E2 469.5126} C_DIS
LIN {X 125.8274,Y -43.3972,Z 166,A -17.2089,B 11.3398,C 0.1415,E1 11.4928,E2 467.6675} C_DIS
LIN {X 127.4129,Y -38.4969,Z 166,A -15.701,B 11.3396,C 0.1545,E1 11.494,E2 466.2448} C_DIS
LIN {X 129.5318,Y -30.6217,Z 166,A -12.1191,B 11.3397,C 0.1425,E1 11.4965,E2 462.6503} C_DIS
LIN {X 130.3661,Y -26.8448,Z 166,A -10.5005,B 11.3397,C 0.1389,E1 11.4974,E2 461.0355} C_DIS
LIN {X 131.0002,Y -23.5549,Z 166,A -9.1704,B 11.3398,C 0.1378,E1 11.4981,E2 459.7175} C_DIS
LIN {X 131.5223,Y -20.4395,Z 166,A -7.7485,B 11.3398,C 0.1321,E1 11.4987,E2 458.2865} C_DIS
LIN {X 132.1161,Y -16.1675,Z 166,A -5.9224,B 11.3399,C 0.1275,E1 11.4994,E2 456.4622} C_DIS
LIN {X 132.4957,Y -12.6807,Z 166,A -4.4304,B 11.3399,C 0.1235,E1 11.4998,E2 454.9707} C_DIS
LIN {X 132.826,Y -8.5627,Z 166,A -2.67,B 11.34,C 0.1188,E1 11.5002,E2 453.2106} C_DIS
LIN {X 133.0068,Y -5.0152,Z 166,A -1.1523,B 11.34,C 0.1146,E1 11.5004,E2 451.6926} C_DIS
LIN {X 133.1005,Y -0.693,Z 166,A 0.5954,B 11.34,C 0.1122,E1 11.5004,E2 449.9568} C_DIS
LIN {X 133.0707,Y 2.9399,Z 166,A 2.2971,B 11.3402,C 0.1039,E1 11.5004,E2 448.2367} C_DIS
LIN {X 132.9229,Y 6.8902,Z 166,A 3.9577,B 11.3402,C 0.1,E1 11.5001,E2 446.5793} C_DIS
LIN {X 132.6325,Y 11.1592,Z 166,A 5.6834,B 11.3402,C 0.0977,E1 11.4998,E2 444.866} C_DIS
LIN {X 132.2612,Y 14.946,Z 166,A 7.3812,B 11.3402,C 0.0913,E1 11.4993,E2 443.1592} C_DIS
LIN {X 131.7949,Y 18.6024,Z 166,A 8.8634,B 11.3402,C 0.0895,E1 11.4987,E2 441.6882} C_DIS
LIN {X 131.2736,Y 21.98,Z 166,A 10.3374,B 11.3403,C 0.0852,E1 11.4981,E2 440.2124} C_DIS
LIN {X 130.5376,Y 26.002,Z 166,A 12.1352,B 11.3403,C 0.0791,E1 11.4971,E2 438.4084} C_DIS
LIN {X 129.7176,Y 29.8199,Z 166,A 13.7725,B 11.3403,C 0.0755,E1 11.4961,E2 436.7748} C_DIS
LIN {X 129.0711,Y 32.5048,Z 166,A 15.5139,B 11.3405,C 0.0572,E1 11.4949,E2 434.9648} C_DIS
LIN {X 127.7476,Y 37.3682,Z 166,A 16.7123,B 11.3404,C 0.0772,E1 11.4941,E2 433.883} C_DIS
LIN {X 126.9389,Y 40.0322,Z 166,A 18.0908,B 11.3404,C 0.0691,E1 11.4929,E2 432.4818} C_DIS
LIN {X 125.9899,Y 42.9287,Z 166,A 19.4479,B 11.3404,C 0.0643,E1 11.4917,E2 431.1181} C_DIS
LIN {X 124.7551,Y 46.3904,Z 166,A 20.8613,B 11.3404,C 0.0644,E1 11.4904,E2 429.7238} C_DIS
LIN {X 123.4228,Y 49.8259,Z 166,A 22.6482,B 11.3404,C 0.0548,E1 11.4885,E2 427.9113} C_DIS
LIN {X 122.0156,Y 53.1801,Z 166,A 24.2965,B 11.3405,C 0.0484,E1 11.4867,E2 426.2518} C_DIS
LIN {X 120.2311,Y 57.0996,Z 166,A 25.8348,B 11.3405,C 0.0519,E1 11.4849,E2 424.7503} C_DIS
LIN {X 117.7205,Y 62.1105,Z 166,A 28.3722,B 11.3405,C 0.0423,E1 11.4817,E2 422.1962} C_DIS
LIN {X 113.9485,Y 68.79,Z 166,A 31.728,B 11.3405,C 0.0327,E1 11.477,E2 418.8319} C_DIS
LIN {X 111.6765,Y 72.4202,Z 166,A 33.5641,B 11.3405,C 0.0283,E1 11.4743,E2 416.9956} C_DIS
LIN {X 109.3684,Y 75.8611,Z 166,A 35.7381,B 11.3406,C 0.0138,E1 11.4708,E2 414.7731} C_DIS
LIN {X 106.8719,Y 79.3395,Z 166,A 37.0606,B 11.3406,C 0.0232,E1 11.4687,E2 413.5127} C_DIS
LIN {X 102.6904,Y 84.6821,Z 166,A 40.0613,B 11.3406,C 0.0145,E1 11.4634,E2 410.5009} C_DIS
LIN {X 99.8325,Y 88.033,Z 166,A 41.9369,B 11.3406,C 0.0109,E1 11.46,E2 408.6269} C_DIS
LIN {X 96.87,Y 91.2826,Z 166,A 43.8157,B 11.3406,C 0.0073,E1 11.4564,E2 406.7489} C_DIS
LIN {X 93.6079,Y 94.6253,Z 166,A 45.7833,B 11.3406,C 0.0043,E1 11.4526,E2 404.7856} C_DIS
LIN {X 90.5431,Y 97.5618,Z 166,A 47.6102,B 11.3406,C 0.0007,E1 11.4489,E2 402.9581} C_DIS
LIN {X 87.2623,Y 100.5072,Z 166,A 49.5093,B 11.3406,C -0.003,E1 11.4449,E2 401.0582} C_DIS
LIN {X 84.2166,Y 103.0721,Z 166,A 51.5676,B 11.3406,C -0.0149,E1 11.4404,E2 398.9578} C_DIS
LIN {X 80.9548,Y 105.6534,Z 166,A 52.9575,B 11.3406,C -0.0078,E1 11.4374,E2 397.6157} C_DIS
LIN {X 77.421,Y 108.2696,Z 166,A 54.6078,B 11.3406,C -0.0048,E1 11.4337,E2 395.9941} C_DIS
LIN {X 73.4822,Y 110.9811,Z 166,A 56.9259,B 11.3406,C -0.0147,E1 11.4283,E2 393.6445} C_DIS
LIN {X 69.7924,Y 113.3375,Z 166,A 58.7199,B 11.3406,C -0.0153,E1 11.4241,E2 391.8611} C_DIS
LIN {X 64.8523,Y 116.2354,Z 166,A 61.2392,B 11.3406,C -0.0201,E1 11.418,E2 389.335} C_DIS
LIN {X 60.7593,Y 118.424,Z 166,A 63.1994,B 11.3406,C -0.0218,E1 11.4131,E2 387.3792} C_DIS
LIN {X 57.2798,Y 120.145,Z 166,A 64.7516,B 11.3406,C -0.0209,E1 11.4093,E2 385.8412} C_DIS
LIN {X 53.8218,Y 121.7347,Z 166,A 66.5027,B 11.3406,C -0.0256,E1 11.4048,E2 384.0766} C_DIS
LIN {X 50.0824,Y 123.3194,Z 166,A 68.1644,B 11.3406,C -0.0253,E1 11.4005,E2 382.4252} C_DIS
LIN {X 46.77,Y 124.6129,Z 166,A 69.6668,B 11.3406,C -0.0262,E1 11.3966,E2 380.9263} C_DIS
LIN {X 43.736,Y 125.71,Z 166,A 71.0486,B 11.3406,C -0.0273,E1 11.393,E2 379.5454} C_DIS
LIN {X 40.9725,Y 126.6385,Z 166,A 72.2758,B 11.3406,C -0.0277,E1 11.3897,E2 378.3218} C_DIS
LIN {X 37.6322,Y 127.6703,Z 166,A 74.0076,B 11.3406,C -0.0344,E1 11.385,E2 376.563} C_DIS
LIN {X 32.9572,Y 128.9562,Z 166,A 75.9326,B 11.3406,C -0.0319,E1 11.3799,E2 374.6578} C_DIS
LIN {X 28.5277,Y 130.0086,Z 166,A 77.909,B 11.3406,C -0.0335,E1 11.3745,E2 372.6799} C_DIS
LIN {X 24.82,Y 130.7664,Z 166,A 79.4841,B 11.3406,C -0.0331,E1 11.3702,E2 371.1117} C_DIS
LIN {X 20.7075,Y 131.4808,Z 166,A 81.3009,B 11.3406,C -0.0343,E1 11.3652,E2 369.293} C_DIS
LIN {X 17.0355,Y 132.0066,Z 166,A 82.9289,B 11.3406,C -0.0356,E1 11.3607,E2 367.6617} C_DIS
LIN {X 13.1675,Y 132.4489,Z 166,A 84.6342,B 11.3406,C -0.0367,E1 11.3559,E2 365.9536} C_DIS
LIN {X 8.7859,Y 132.8122,Z 166,A 86.5015,B 11.3406,C -0.0364,E1 11.3507,E2 364.0901} C_DIS
LIN {X 5.3223,Y 132.9948,Z 166,A 87.8695,B 11.3406,C -0.0336,E1 11.347,E2 362.7375} C_DIS
LIN {X 1.9739,Y 133.0868,Z 166,A 89.3274,B 11.3406,C -0.034,E1 11.3429,E2 361.2783} C_DIS
LIN {X -1.9474,Y 133.0872,Z 166,A 91.0674,B 11.3406,C -0.0351,E1 11.338,E2 359.5329} C_DIS
LIN {X -6.0039,Y 132.9674,Z 166,A 92.8909,B 11.3406,C -0.0366,E1 11.3329,E2 357.7012} C_DIS
LIN {X -9.8191,Y 132.7385,Z 166,A 94.4765,B 11.3406,C -0.0348,E1 11.3285,E2 356.1236} C_DIS
LIN {X -13.882,Y 132.3757,Z 166,A 96.2459,B 11.3406,C -0.0345,E1 11.3236,E2 354.3536} C_DIS
LIN {X -17.6657,Y 131.924,Z 166,A 97.9228,B 11.3406,C -0.0347,E1 11.3189,E2 352.6733} C_DIS
LIN {X -21.7713,Y 131.3084,Z 166,A 99.6294,B 11.3406,C -0.0319,E1 11.3142,E2 350.9774} C_DIS
LIN {X -25.7945,Y 130.5798,Z 166,A 102.4636,B 11.3405,C -0.0555,E1 11.3062,E2 348.0157} C_DIS
LIN {X -32.8358,Y 128.987,Z 166,A 104.4964,B 11.3405,C -0.0286,E1 11.301,E2 346.1139} C_DIS
LIN {X -35.7242,Y 128.2171,Z 166,A 106.784,B 11.3405,C -0.0502,E1 11.2946,E2 343.7076} C_DIS
LIN {X -42.2559,Y 126.2153,Z 166,A 108.5231,B 11.3406,C -0.0202,E1 11.2903,E2 342.1144} C_DIS
LIN {X -44.7614,Y 125.3491,Z 166,A 109.9491,B 11.3406,C -0.0254,E1 11.2864,E2 340.6556} C_DIS
LIN {X -47.8317,Y 124.2099,Z 166,A 111.3297,B 11.3406,C -0.0232,E1 11.2828,E2 339.2796} C_DIS
LIN {X -52.0035,Y 122.5235,Z 166,A 113.7079,B 11.3406,C -0.0307,E1 11.2766,E2 336.8506} C_DIS
LIN {X -55.5669,Y 120.9472,Z 166,A 115.2014,B 11.3406,C -0.0245,E1 11.2729,E2 335.3803} C_DIS
LIN {X -59.3472,Y 119.1384,Z 166,A 117.1612,B 11.3406,C -0.0255,E1 11.2679,E2 333.4035} C_DIS
LIN {X -62.7535,Y 117.3809,Z 166,A 118.8183,B 11.3406,C -0.0233,E1 11.2638,E2 331.7471} C_DIS
LIN {X -66.0441,Y 115.5617,Z 166,A 120.1221,B 11.3406,C -0.014,E1 11.2608,E2 330.4824} C_DIS
LIN {X -69.9266,Y 113.2551,Z 166,A 122.1221,B 11.3406,C -0.0121,E1 11.256,E2 328.4776} C_DIS
LIN {X -73.6667,Y 110.8585,Z 166,A 124.0537,B 11.3406,C -0.0094,E1 11.2514,E2 326.5455} C_DIS
LIN {X -77.1966,Y 108.43,Z 166,A 125.9171,B 11.3406,C -0.0066,E1 11.2472,E2 324.6816} C_DIS
LIN {X -80.8998,Y 105.6955,Z 166,A 127.8826,B 11.3406,C -0.0026,E1 11.2428,E2 322.72} C_DIS
LIN {X -84.3522,Y 102.9613,Z 166,A 129.8055,B 11.3406,C 0.0004,E1 11.2386,E2 320.7958} C_DIS
LIN {X -87.8306,Y 100.0113,Z 166,A 131.8228,B 11.3406,C 0.0031,E1 11.2343,E2 318.7741} C_DIS
LIN {X -91.1693,Y 96.9769,Z 166,A 133.7487,B 11.3406,C 0.0074,E1 11.2304,E2 316.8522} C_DIS
LIN {X -94.333,Y 93.9021,Z 166,A 135.6705,B 11.3406,C 0.0109,E1 11.2266,E2 314.9296} C_DIS
LIN {X -97.5687,Y 90.5357,Z 166,A 137.6621,B 11.3406,C 0.0157,E1 11.2228,E2 312.9424} C_DIS
LIN {X -100.462,Y 87.3142,Z 166,A 139.5387,B 11.3406,C 0.0196,E1 11.2193,E2 311.0663} C_DIS
LIN {X -103.1549,Y 84.1154,Z 166,A 141.3841,B 11.3406,C 0.0228,E1 11.216,E2 309.2175} C_DIS
LIN {X -105.952,Y 80.5644,Z 166,A 143.3798,B 11.3406,C 0.0264,E1 11.2126,E2 307.2181} C_DIS
LIN {X -108.5537,Y 77.023,Z 166,A 145.2984,B 11.3406,C 0.0304,E1 11.2095,E2 305.2983} C_DIS
LIN {X -111.2491,Y 73.0751,Z 166,A 148.0588,B 11.3406,C 0.0208,E1 11.2051,E2 302.4561} C_DIS
LIN {X -114.3351,Y 68.1454,Z 166,A 150.0414,B 11.3406,C 0.0381,E1 11.2023,E2 300.5389} C_DIS
LIN {X -116.8185,Y 63.7946,Z 166,A 151.9688,B 11.3406,C 0.0485,E1 11.1997,E2 298.6413} C_DIS
LIN {X -118.3255,Y 60.9529,Z 166,A 153.3843,B 11.3406,C 0.0515,E1 11.1979,E2 297.2236} C_DIS
LIN {X -120.5042,Y 56.5247,Z 166,A 155.4778,B 11.3405,C 0.0578,E1 11.1954,E2 295.1363} C_DIS
LIN {X -121.7868,Y 53.7034,Z 166,A 157.1563,B 11.3405,C 0.0543,E1 11.1934,E2 293.4182} C_DIS
LIN {X -123.9041,Y 48.6185,Z 166,A 159.348,B 11.3405,C 0.0646,E1 11.1912,E2 291.2506} C_DIS
LIN {X -125.2501,Y 45.0359,Z 166,A 160.9437,B 11.3405,C 0.0702,E1 11.1896,E2 289.663} C_DIS
LIN {X -126.4608,Y 41.5188,Z 166,A 162.6714,B 11.3405,C 0.0721,E1 11.1881,E2 287.9221} C_DIS
LIN {X -127.6827,Y 37.5899,Z 166,A 164.3116,B 11.3403,C 0.0798,E1 11.1868,E2 286.2995} C_DIS
LIN {X -128.6014,Y 34.3149,Z 166,A 165.851,B 11.3403,C 0.0825,E1 11.1856,E2 284.7528} C_DIS
LIN {X -129.7771,Y 29.5596,Z 166,A 168.1525,B 11.3403,C 0.0846,E1 11.1841,E2 282.4306} C_DIS
LIN {X -130.6064,Y 25.6572,Z 166,A 170.2527,B 11.3403,C 0.0817,E1 11.183,E2 280.2864} C_DIS
LIN {X -131.3678,Y 21.4093,Z 166,A 171.9114,B 11.3403,C 0.0912,E1 11.1822,E2 278.6536} C_DIS
LIN {X -131.8736,Y 18.0464,Z 166,A 173.0977,B 11.3402,C 0.1012,E1 11.1818,E2 277.5023} C_DIS
LIN {X -132.3443,Y 14.1733,Z 166,A 174.7847,B 11.3402,C 0.106,E1 11.1812,E2 275.8161} C_DIS
LIN {X -132.6963,Y 10.3979,Z 166,A 176.6073,B 11.3402,C 0.1069,E1 11.1808,E2 273.9726} C_DIS
LIN {X -132.9732,Y 5.8752,Z 166,A 178.4485,B 11.3401,C 0.1149,E1 11.1805,E2 272.1466} C_DIS
LIN {X -133.0856,Y 2.0488,Z 166,A -179.8858,B 11.3401,C 0.1193,E1 11.1805,E2 270.4805} C_DIS
LIN {X -133.0815,Y -2.2936,Z 166,A -177.9774,B 11.34,C 0.124,E1 11.1805,E2 268.5694} C_DIS
LIN {X -132.9544,Y -6.2621,Z 166,A -176.2377,B 11.34,C 0.1284,E1 11.1807,E2 266.8277} C_DIS
LIN {X -132.7123,Y -10.1785,Z 166,A -174.4319,B 11.3399,C 0.131,E1 11.181,E2 265.0097} C_DIS
LIN {X -132.3219,Y -14.382,Z 166,A -172.7166,B 11.3398,C 0.1384,E1 11.1815,E2 263.3083} C_DIS
LIN {X -131.8684,Y -18.0881,Z 166,A -171.0221,B 11.3398,C 0.1412,E1 11.1821,E2 261.605} C_DIS
LIN {X -131.1333,Y -22.8113,Z 166,A -168.7073,B 11.3398,C 0.1419,E1 11.1832,E2 259.2612} C_DIS
LIN {X -129.9144,Y -28.9585,Z 166,A -166.1648,B 11.3396,C 0.1528,E1 11.1846,E2 256.7399} C_DIS
LIN {X -129.1052,Y -32.3701,Z 166,A -163.9084,B 11.3398,C 0.1415,E1 11.1863,E2 254.3941} C_DIS
LIN {X -127.4912,Y -38.2408,Z 166,A -162.0419,B 11.3394,C 0.1646,E1 11.1876,E2 252.6217} C_DIS
LIN {X -126.3217,Y -41.9363,Z 166,A -160.4032,B 11.3394,C 0.1698,E1 11.189,E2 250.9879} C_DIS
LIN {X -125.1229,Y -45.3887,Z 166,A -158.7986,B 11.3394,C 0.1735,E1 11.1905,E2 249.3809} C_DIS
LIN {X -123.6559,Y -49.2477,Z 166,A -156.9342,B 11.3393,C 0.1765,E1 11.1924,E2 247.5074} C_DIS
LIN {X -122.2016,Y -52.75,Z 166,A -155.6039,B 11.3391,C 0.1871,E1 11.1938,E2 246.2148} C_DIS
LIN {X -121.2605,Y -54.8819,Z 166,A -154.35,B 11.3391,C 0.1845,E1 11.1953,E2 244.9315} C_DIS
LIN {X -119.1086,Y -59.4076,Z 166,A -152.1607,B 11.3391,C 0.1895,E1 11.198,E2 242.7399} C_DIS
LIN {X -117.2191,Y -63.0555,Z 166,A -150.2782,B 11.3391,C 0.1916,E1 11.2004,E2 240.8449} C_DIS
LIN {X -115.0346,Y -66.9586,Z 166,A -148.3181,B 11.339,C 0.1957,E1 11.2032,E2 238.8819} C_DIS
LIN {X -112.8893,Y -70.515,Z 166,A -146.801,B 11.3388,C 0.2058,E1 11.2053,E2 237.3987} C_DIS
LIN {X -110.4791,Y -74.2347,Z 166,A -144.6737,B 11.3388,C 0.2058,E1 11.2086,E2 235.2462} C_DIS
LIN {X -108.3948,Y -77.2458,Z 166,A -143.1133,B 11.3388,C 0.2098,E1 11.2111,E2 233.6886} C_DIS
LIN {X -106.1934,Y -80.2451,Z 166,A -141.4699,B 11.3387,C 0.2125,E1 11.2139,E2 232.041} C_DIS
LIN {X -103.8487,Y -83.2581,Z 166,A -139.6791,B 11.3387,C 0.213,E1 11.217,E2 230.2332} C_DIS
LIN {X -100.9909,Y -86.7017,Z 166,A -137.6693,B 11.3387,C 0.2154,E1 11.2206,E2 228.2141} C_DIS
LIN {X -97.6812,Y -90.4149,Z 166,A -135.6061,B 11.3385,C 0.2216,E1 11.2245,E2 226.1615} C_DIS
LIN {X -94.6744,Y -93.5585,Z 166,A -133.6962,B 11.3385,C 0.2246,E1 11.2282,E2 224.2477} C_DIS
LIN {X -91.639,Y -96.5337,Z 166,A -131.838,B 11.3384,C 0.2275,E1 11.232,E2 222.3868} C_DIS
LIN {X -87.9774,Y -99.8816,Z 166,A -129.4949,B 11.3384,C 0.2269,E1 11.2369,E2 220.019} C_DIS
LIN {X -85.4393,Y -102.0608,Z 166,A -128.0506,B 11.3384,C 0.2294,E1 11.24,E2 218.5747} C_DIS
LIN {X -82.8542,Y -104.1705,Z 166,A -126.8324,B 11.3382,C 0.2368,E1 11.2426,E2 217.3836} C_DIS
LIN {X -79.29,Y -106.9087,Z 166,A -124.9459,B 11.3381,C 0.2411,E1 11.2468,E2 215.5034} C_DIS
LIN {X -75.8411,Y -109.3823,Z 166,A -123.051,B 11.3381,C 0.2425,E1 11.2511,E2 213.6007} C_DIS
LIN {X -72.1739,Y -111.8363,Z 166,A -121.1729,B 11.338,C 0.2458,E1 11.2555,E2 211.7255} C_DIS
LIN {X -67.7777,Y -114.5541,Z 166,A -118.8341,B 11.338,C 0.2464,E1 11.2611,E2 209.3731} C_DIS
LIN {X -64.1121,Y -116.6452,Z 166,A -117.1742,B 11.3379,C 0.2524,E1 11.2651,E2 207.7326} C_DIS
LIN {X -60.8611,Y -118.3722,Z 166,A -115.4077,B 11.3379,C 0.2502,E1 11.2695,E2 205.9438} C_DIS
LIN {X -57.2062,Y -120.1802,Z 166,A -113.8388,B 11.3378,C 0.2565,E1 11.2734,E2 204.3978} C_DIS
LIN {X -54.8376,Y -121.2803,Z 166,A -112.6053,B 11.3378,C 0.2553,E1 11.2766,E2 203.151} C_DIS
LIN {X -51.2348,Y -122.8446,Z 166,A -110.9609,B 11.3378,C 0.2581,E1 11.2808,E2 201.5122} C_DIS
LIN {X -48.1065,Y -124.1031,Z 166,A -109.4543,B 11.3378,C 0.2581,E1 11.2847,E2 199.9987} C_DIS
LIN {X -44.0443,Y -125.6031,Z 166,A -107.5936,B 11.3377,C 0.2599,E1 11.2896,E2 198.1383} C_DIS
LIN {X -40.9373,Y -126.6498,Z 166,A -106.0334,B 11.3377,C 0.2576,E1 11.2938,E2 196.5597} C_DIS
LIN {X -36.3392,Y -128.0451,Z 166,A -103.9498,B 11.3377,C 0.2587,E1 11.2994,E2 194.4738} C_DIS
LIN {X -31.5654,Y -129.3044,Z 166,A -101.9812,B 11.3377,C 0.2636,E1 11.3047,E2 192.5241} C_DIS
LIN {X -28.0975,Y -130.1014,Z 166,A -100.5094,B 11.3376,C 0.2658,E1 11.3087,E2 191.0593} C_DIS
LIN {X -25.4607,Y -130.644,Z 166,A -99.2701,B 11.3376,C 0.2644,E1 11.3121,E2 189.8098} C_DIS
LIN {X -21.9742,Y -131.2746,Z 166,A -97.7744,B 11.3376,C 0.2657,E1 11.3162,E2 188.3173} C_DIS
LIN {X -17.9626,Y -131.8851,Z 166,A -95.9367,B 11.3376,C 0.264,E1 11.3213,E2 186.4679} C_DIS
LIN {X -14.1847,Y -132.3431,Z 166,A -94.3702,B 11.3376,C 0.2661,E1 11.3256,E2 184.9095} C_DIS
LIN {X -10.2542,Y -132.7067,Z 166,A -92.6285,B 11.3376,C 0.2653,E1 11.3305,E2 183.162} C_DIS
LIN {X -6.4604,Y -132.9445,Z 166,A -91.0454,B 11.3376,C 0.2666,E1 11.3349,E2 181.5847} C_DIS
LIN {X -2.3641,Y -133.0803,Z 166,A -89.2807,B 11.3376,C 0.2665,E1 11.3398,E2 179.8192} C_DIS
LIN {X 0.9656,Y -133.095,Z 166,A -88.395,B 11.3372,C 0.2795,E1 11.3421,E2 178.9998} C_DIS
Enddeposition()
LIN {X 0.9656,Y -133.095,Z 166,A -88.395,B 11.3372,C 0.2795,E1 11.3421,E2 178.9998} C_DIS
Startdeposition()
$VEL.CP = VEL_PRINT
LIN {X -1.1358,Y -134.0134,Z 166,A -89.4119,B 11.1387,C 0.2986,E1 11.141,E2 180.1259} C_DIS
LIN {X -5.5942,Y -133.9013,Z 166,A -91.1934,B 11.1387,C 0.2957,E1 11.136,E2 181.8929} C_DIS
LIN {X -9.3308,Y -133.693,Z 166,A -92.8756,B 11.1387,C 0.2976,E1 11.1313,E2 183.5859} C_DIS
LIN {X -12.7994,Y -133.4049,Z 166,A -94.3035,B 11.1387,C 0.296,E1 11.1274,E2 185.007} C_DIS
LIN {X -16.2224,Y -133.0325,Z 166,A -95.7783,B 11.1387,C 0.2957,E1 11.1233,E2 186.4826} C_DIS
LIN {X -19.8707,Y -132.5377,Z 166,A -97.4282,B 11.1387,C 0.297,E1 11.1187,E2 188.1424} C_DIS
LIN {X -23.5181,Y -131.9377,Z 166,A -98.9301,B 11.1388,C 0.2946,E1 11.1146,E2 189.6351} C_DIS
LIN {X -27.2077,Y -131.2274,Z 166,A -100.5155,B 11.1388,C 0.2934,E1 11.1102,E2 191.2183} C_DIS
LIN {X -30.0607,Y -130.6026,Z 166,A -101.8359,B 11.1388,C 0.2945,E1 11.1066,E2 192.5479} C_DIS
LIN {X -35.2837,Y -129.2915,Z 166,A -104.0961,B 11.1388,C 0.2921,E1 11.1005,E2 194.8034} C_DIS
LIN {X -38.1182,Y -128.4829,Z 166,A -105.4923,B 11.1388,C 0.2943,E1 11.0967,E2 196.2164} C_DIS
LIN {X -42.0247,Y -127.2582,Z 166,A -107.2791,B 11.1388,C 0.2938,E1 11.092,E2 198.0079} C_DIS
LIN {X -45.7867,Y -125.9536,Z 166,A -108.8628,B 11.1389,C 0.2896,E1 11.0878,E2 199.5773} C_DIS
LIN {X -49.0861,Y -124.7055,Z 166,A -110.3347,B 11.1389,C 0.2874,E1 11.084,E2 201.0449} C_DIS
LIN {X -51.8343,Y -123.5873,Z 166,A -111.6149,B 11.139,C 0.2864,E1 11.0807,E2 202.3265} C_DIS
LIN {X -54.763,Y -122.3176,Z 166,A -113.0436,B 11.139,C 0.2864,E1 11.077,E2 203.7631} C_DIS
LIN {X -58.4649,Y -120.5944,Z 166,A -114.8747,B 11.139,C 0.2863,E1 11.0724,E2 205.6046} C_DIS
LIN {X -61.2511,Y -119.202,Z 166,A -116.1955,B 11.139,C 0.2844,E1 11.0691,E2 206.924} C_DIS
LIN {X -65.3016,Y -117.0341,Z 166,A -118.1577,B 11.1391,C 0.2818,E1 11.0643,E2 208.8859} C_DIS
LIN {X -69.7568,Y -114.4344,Z 166,A -120.4437,B 11.1391,C 0.2805,E1 11.0588,E2 211.1814} C_DIS
LIN {X -73.7843,Y -111.8794,Z 166,A -122.4328,B 11.1393,C 0.2764,E1 11.0541,E2 213.1641} C_DIS
LIN {X -77.5398,Y -109.3106,Z 166,A -124.3979,B 11.1393,C 0.2738,E1 11.0496,E2 215.1312} C_DIS
LIN {X -80.8304,Y -106.8998,Z 166,A -126.1299,B 11.1394,C 0.2706,E1 11.0458,E2 216.8613} C_DIS
LIN {X -84.3492,Y -104.1459,Z 166,A -128.6249,B 11.1392,C 0.2798,E1 11.0402,E2 219.4264} C_DIS
LIN {X -88.1659,Y -100.935,Z 166,A -130.0711,B 11.1396,C 0.2613,E1 11.0373,E2 220.7891} C_DIS
LIN {X -90.8931,Y -98.4866,Z 166,A -131.8248,B 11.1396,C 0.2623,E1 11.0336,E2 222.5649} C_DIS
LIN {X -94.0551,Y -95.4716,Z 166,A -133.7107,B 11.1396,C 0.259,E1 11.0298,E2 224.4523} C_DIS
LIN {X -97.2057,Y -92.2622,Z 166,A -135.689,B 11.1397,C 0.2563,E1 11.026,E2 226.4365} C_DIS
LIN {X -100.9215,Y -88.1814,Z 166,A -137.8395,B 11.14,C 0.2469,E1 11.022,E2 228.5607} C_DIS
LIN {X -103.2388,Y -85.4568,Z 166,A -139.5692,B 11.14,C 0.2478,E1 11.0189,E2 230.3139} C_DIS
LIN {X -105.9658,Y -82.0509,Z 166,A -141.5219,B 11.14,C 0.2455,E1 11.0155,E2 232.2762} C_DIS
LIN {X -108.8003,Y -78.2543,Z 166,A -143.5227,B 11.14,C 0.2403,E1 11.0122,E2 234.2729} C_DIS
LIN {X -112.0862,Y -73.4693,Z 166,A -146.0316,B 11.1402,C 0.235,E1 11.0083,E2 236.7835} C_DIS
LIN {X -114.4298,Y -69.7643,Z 166,A -147.8772,B 11.1403,C 0.2298,E1 11.0055,E2 238.6245} C_DIS
LIN {X -116.6194,Y -66.0394,Z 166,A -149.786,B 11.1403,C 0.2265,E1 11.0029,E2 240.5395} C_DIS
LIN {X -118.6485,Y -62.3145,Z 166,A -151.5704,B 11.1405,C 0.2213,E1 11.0005,E2 242.319} C_DIS
LIN {X -120.6596,Y -58.3265,Z 166,A -153.7401,B 11.1405,C 0.2217,E1 10.9978,E2 244.5187} C_DIS
LIN {X -122.0613,Y -55.3359,Z 166,A -155.0674,B 11.1405,C 0.2162,E1 10.9963,E2 245.8349} C_DIS
LIN {X -123.7282,Y -51.497,Z 166,A -156.6824,B 11.1407,C 0.2079,E1 10.9945,E2 247.4274} C_DIS
LIN {X -124.9908,Y -48.3523,Z 166,A -158.1364,B 11.1408,C 0.2041,E1 10.9931,E2 248.881} C_DIS
LIN {X -126.0614,Y -45.4876,Z 166,A -159.4852,B 11.1408,C 0.2014,E1 10.9918,E2 250.2336} C_DIS
LIN {X -127.1926,Y -42.2215,Z 166,A -160.9982,B 11.1409,C 0.198,E1 10.9904,E2 251.7496} C_DIS
LIN {X -128.3963,Y -38.414,Z 166,A -164.0528,B 11.1405,C 0.2203,E1 10.9879,E2 254.9627} C_DIS
LIN {X -130.5909,Y -30.1122,Z 166,A -166.2045,B 11.1412,C 0.1795,E1 10.9866,E2 256.9308} C_DIS
LIN {X -131.929,Y -23.5672,Z 166,A -169.2875,B 11.1412,C 0.176,E1 10.9849,E2 260.0386} C_DIS
LIN {X -132.6815,Y -18.876,Z 166,A -171.3473,B 11.1414,C 0.1707,E1 10.984,E2 262.1} C_DIS
LIN {X -133.0958,Y -15.6916,Z 166,A -172.7996,B 11.1414,C 0.1683,E1 10.9835,E2 263.5604} C_DIS
LIN {X -133.5213,Y -11.5251,Z 166,A -174.641,B 11.1414,C 0.1641,E1 10.983,E2 265.4061} C_DIS
LIN {X -133.806,Y -7.5583,Z 166,A -176.4575,B 11.1415,C 0.1615,E1 10.9826,E2 267.2349} C_DIS
LIN {X -133.9684,Y -3.6335,Z 166,A -178.0159,B 11.1416,C 0.1541,E1 10.9825,E2 268.7771} C_DIS
LIN {X -134.0206,Y 0.1602,Z 166,A -179.8335,B 11.1416,C 0.1533,E1 10.9825,E2 270.6165} C_DIS
LIN {X -133.9428,Y 4.5309,Z 166,A 178.2884,B 11.1416,C 0.1479,E1 10.9826,E2 272.4936} C_DIS
LIN {X -133.7413,Y 8.6091,Z 166,A 176.6784,B 11.1418,C 0.1401,E1 10.9829,E2 274.0855} C_DIS
LIN {X -133.4246,Y 12.5938,Z 166,A 174.9159,B 11.1418,C 0.1362,E1 10.9833,E2 275.8527} C_DIS
LIN {X -133.0216,Y 16.3135,Z 166,A 173.2312,B 11.1418,C 0.1332,E1 10.9838,E2 277.5457} C_DIS
LIN {X -131.7706,Y 24.4478,Z 166,A 169.8038,B 11.142,C 0.1211,E1 10.9853,E2 280.9586} C_DIS
LIN {X -131.0847,Y 27.8857,Z 166,A 168.1381,B 11.142,C 0.1201,E1 10.9863,E2 282.6424} C_DIS
LIN {X -130.1278,Y 32.0598,Z 166,A 166.3195,B 11.142,C 0.1146,E1 10.9875,E2 284.4575} C_DIS
LIN {X -129.3434,Y 35.0891,Z 166,A 165.0597,B 11.1421,C 0.1092,E1 10.9883,E2 285.7066} C_DIS
LIN {X -128.5163,Y 38.0039,Z 166,A 163.7478,B 11.1421,C 0.1059,E1 10.9894,E2 287.0189} C_DIS
LIN {X -127.6121,Y 40.9364,Z 166,A 162.4134,B 11.1421,C 0.1026,E1 10.9905,E2 288.3545} C_DIS
LIN {X -126.5697,Y 44.0539,Z 166,A 160.9989,B 11.1422,C 0.0989,E1 10.9918,E2 289.7685} C_DIS
LIN {X -125.4928,Y 47.0334,Z 166,A 159.564,B 11.1422,C 0.0967,E1 10.9931,E2 291.2114} C_DIS
LIN {X -124.2197,Y 50.3,Z 166,A 158.0321,B 11.1422,C 0.0932,E1 10.9947,E2 292.7455} C_DIS
LIN {X -122.0629,Y 55.3324,Z 166,A 155.7284,B 11.1423,C 0.0861,E1 10.9973,E2 295.0424} C_DIS
LIN {X -120.8236,Y 57.9852,Z 166,A 154.3883,B 11.1423,C 0.0845,E1 10.9989,E2 296.3914} C_DIS
LIN {X -119.3198,Y 61.0197,Z 166,A 152.9706,B 11.1423,C 0.0801,E1 11.0007,E2 297.8039} C_DIS
LIN {X -117.6541,Y 64.1765,Z 166,A 151.3452,B 11.1423,C 0.0781,E1 11.0028,E2 299.4394} C_DIS
LIN {X -115.3884,Y 68.1669,Z 166,A 149.388,B 11.1424,C 0.073,E1 11.0056,E2 301.3939} C_DIS
LIN {X -112.176,Y 73.3336,Z 166,A 146.7887,B 11.1424,C 0.0664,E1 11.0094,E2 303.9901} C_DIS
LIN {X -109.8502,Y 76.7732,Z 166,A 144.8936,B 11.1424,C 0.0644,E1 11.0125,E2 305.8974} C_DIS
LIN {X -107.2065,Y 80.424,Z 166,A 142.9501,B 11.1424,C 0.0602,E1 11.0157,E2 307.8407} C_DIS
LIN {X -104.5137,Y 83.8933,Z 166,A 141.029,B 11.1425,C 0.0566,E1 11.019,E2 309.7649} C_DIS
LIN {X -101.5702,Y 87.4334,Z 166,A 139.0761,B 11.1425,C 0.0518,E1 11.0225,E2 311.7138} C_DIS
LIN {X -98.5467,Y 90.8277,Z 166,A 137.1468,B 11.1425,C 0.0472,E1 11.0261,E2 313.6394} C_DIS
LIN {X -95.4765,Y 94.0501,Z 166,A 135.2136,B 11.1425,C 0.0437,E1 11.0299,E2 315.5742} C_DIS
LIN {X -92.3788,Y 97.0945,Z 166,A 133.3111,B 11.1425,C 0.0408,E1 11.0337,E2 317.4801} C_DIS
LIN {X -89.2078,Y 100.0157,Z 166,A 131.4639,B 11.1425,C 0.0372,E1 11.0375,E2 319.3259} C_DIS
LIN {X -85.9825,Y 102.8015,Z 166,A 129.6223,B 11.1426,C 0.034,E1 11.0414,E2 321.1679} C_DIS
LIN {X -82.4778,Y 105.6345,Z 166,A 127.6419,B 11.1426,C 0.0316,E1 11.0458,E2 323.1527} C_DIS
LIN {X -78.8711,Y 108.3537,Z 166,A 125.7598,B 11.1426,C 0.0271,E1 11.05,E2 325.0271} C_DIS
LIN {X -75.6345,Y 110.6372,Z 166,A 124.0255,B 11.1426,C 0.025,E1 11.054,E2 326.7645} C_DIS
LIN {X -71.9975,Y 113.0379,Z 166,A 122.1423,B 11.1426,C 0.0224,E1 11.0584,E2 328.6484} C_DIS
LIN {X -68.3241,Y 115.2955,Z 166,A 120.261,B 11.1426,C 0.0203,E1 11.0629,E2 330.5325} C_DIS
LIN {X -61.0672,Y 119.2957,Z 166,A 117.0245,B 11.1426,C 0.0086,E1 11.0707,E2 333.7296} C_DIS
LIN {X -57.4146,Y 121.0962,Z 166,A 115.0595,B 11.1426,C 0.0111,E1 11.0757,E2 335.7196} C_DIS
LIN {X -53.6063,Y 122.8298,Z 166,A 113.1061,B 11.1426,C 0.0124,E1 11.0807,E2 337.6909} C_DIS
LIN {X -49.9679,Y 124.3536,Z 166,A 111.5205,B 11.1426,C 0.0083,E1 11.0848,E2 339.2632} C_DIS
LIN {X -46.5217,Y 125.6845,Z 166,A 110.0032,B 11.1426,C 0.0052,E1 11.0887,E2 340.7719} C_DIS
LIN {X -43.7361,Y 126.6799,Z 166,A 108.6857,B 11.1426,C 0.0051,E1 11.0922,E2 342.0947} C_DIS
LIN {X -36.4665,Y 128.9611,Z 166,A 105.3236,B 11.1426,C 0.0044,E1 11.1013,E2 345.4668} C_DIS
LIN {X -32.4537,Y 130.0295,Z 166,A 102.6741,B 11.1426,C 0.0222,E1 11.1087,E2 348.2173} C_DIS
LIN {X -25.7899,Y 131.514,Z 166,A 100.8082,B 11.1426,C -0.0028,E1 11.1135,E2 349.958} C_DIS
LIN {X -21.0786,Y 132.3507,Z 166,A 98.5639,B 11.1426,C 0.0005,E1 11.1197,E2 352.2245} C_DIS
LIN {X -17.2807,Y 132.8987,Z 166,A 97.0059,B 11.1426,C -0.0021,E1 11.124,E2 353.7718} C_DIS
LIN {X -13.4022,Y 133.347,Z 166,A 95.2648,B 11.1426,C -0.0011,E1 11.1288,E2 355.5204} C_DIS
LIN {X -9.6197,Y 133.6719,Z 166,A 93.7642,B 11.1426,C -0.0043,E1 11.133,E2 357.0056} C_DIS
LIN {X -6.2309,Y 133.8736,Z 166,A 92.1806,B 11.1426,C -0.0016,E1 11.1374,E2 358.6042} C_DIS
LIN {X -1.985,Y 134.0032,Z 166,A 90.4692,B 11.1426,C -0.0042,E1 11.1422,E2 360.3023} C_DIS
LIN {X 1.4671,Y 134.0116,Z 166,A 88.8616,B 11.1426,C -0.0013,E1 11.1467,E2 361.9249} C_DIS
LIN {X 5.3612,Y 133.9104,Z 166,A 87.3709,B 11.1426,C -0.0052,E1 11.1508,E2 363.3942} C_DIS
LIN {X 9.0166,Y 133.7159,Z 166,A 85.6302,B 11.1426,C -0.0009,E1 11.1557,E2 365.1551} C_DIS
LIN {X 12.8902,Y 133.3962,Z 166,A 84.0521,B 11.1426,C -0.0025,E1 11.1601,E2 366.7226} C_DIS
LIN {X 17.4001,Y 132.8831,Z 166,A 82.1046,B 11.1426,C -0.0018,E1 11.1655,E2 368.6703} C_DIS
LIN {X 21.73,Y 132.2444,Z 166,A 80.2171,B 11.1426,C -0.0007,E1 11.1707,E2 370.5591} C_DIS
LIN {X 25.3127,Y 131.6052,Z 166,A 78.753,B 11.1426,C -0.0021,E1 11.1747,E2 372.0119} C_DIS
LIN {X 28.978,Y 130.8489,Z 166,A 76.824,B 11.1426,C 0.0066,E1 11.18,E2 373.9795} C_DIS
LIN {X 32.27,Y 130.0761,Z 166,A 75.7526,B 11.1426,C -0.0013,E1 11.1828,E2 375.0064} C_DIS
LIN {X 34.9367,Y 129.384,Z 166,A 74.3971,B 11.1426,C 0.0037,E1 11.1865,E2 376.3827} C_DIS
LIN {X 39.0236,Y 128.21,Z 166,A 72.5601,B 11.1426,C 0.0056,E1 11.1915,E2 378.2217} C_DIS
LIN {X 44.1355,Y 126.5414,Z 166,A 70.4792,B 11.1426,C 0.0024,E1 11.1969,E2 380.2765} C_DIS
LIN {X 47.1666,Y 125.443,Z 166,A 69.0554,B 11.1426,C 0.0049,E1 11.2006,E2 381.7056} C_DIS
LIN {X 50.2294,Y 124.2482,Z 166,A 67.6401,B 11.1426,C 0.0065,E1 11.2043,E2 383.1219} C_DIS
LIN {X 53.8119,Y 122.7409,Z 166,A 66.023,B 11.1426,C 0.0073,E1 11.2085,E2 384.7337} C_DIS
LIN {X 56.8201,Y 121.3773,Z 166,A 64.6162,B 11.1426,C 0.0089,E1 11.212,E2 386.1399} C_DIS
LIN {X 59.8887,Y 119.8931,Z 166,A 63.0871,B 11.1426,C 0.0124,E1 11.2159,E2 387.6776} C_DIS
LIN {X 63.7403,Y 117.8915,Z 166,A 61.0427,B 11.1426,C 0.0195,E1 11.221,E2 389.7446} C_DIS
LIN {X 69.1504,Y 114.8015,Z 166,A 58.7873,B 11.1426,C 0.0133,E1 11.2263,E2 391.9516} C_DIS
LIN {X 71.7983,Y 113.1645,Z 166,A 57.2771,B 11.1426,C 0.0197,E1 11.2299,E2 393.4835} C_DIS
LIN {X 75.2634,Y 110.8898,Z 166,A 55.0709,B 11.1426,C 0.0333,E1 11.2352,E2 395.7416} C_DIS
LIN {X 78.8503,Y 108.3688,Z 166,A 53.8804,B 11.1426,C 0.0194,E1 11.2377,E2 396.8511} C_DIS
LIN {X 80.991,Y 106.7783,Z 166,A 52.0169,B 11.1426,C 0.0394,E1 11.242,E2 398.801} C_DIS
LIN {X 84.687,Y 103.8713,Z 166,A 50.8092,B 11.1426,C 0.023,E1 11.2445,E2 399.9138} C_DIS
LIN {X 87.016,Y 101.9284,Z 166,A 49.2056,B 11.1426,C 0.0331,E1 11.248,E2 401.5546} C_DIS
LIN {X 90.3982,Y 98.9416,Z 166,A 47.2626,B 11.1426,C 0.0372,E1 11.252,E2 403.4998} C_DIS
LIN {X 93.6639,Y 95.8553,Z 166,A 45.3745,B 11.1426,C 0.0401,E1 11.2558,E2 405.3848} C_DIS
LIN {X 96.6918,Y 92.8002,Z 166,A 43.5455,B 11.1426,C 0.0437,E1 11.2594,E2 407.2134} C_DIS
LIN {X 99.8392,Y 89.4049,Z 166,A 41.6242,B 11.1426,C 0.0464,E1 11.263,E2 409.1286} C_DIS
LIN {X 102.8126,Y 85.9693,Z 166,A 39.6935,B 11.1426,C 0.0504,E1 11.2665,E2 411.0588} C_DIS
LIN {X 107.0241,Y 80.6657,Z 166,A 36.9053,B 11.1426,C 0.0542,E1 11.2712,E2 413.8357} C_DIS
LIN {X 110.3866,Y 75.9996,Z 166,A 34.3906,B 11.1425,C 0.0615,E1 11.2753,E2 416.3586} C_DIS
LIN {X 112.8705,Y 72.2589,Z 166,A 32.5316,B 11.1425,C 0.0646,E1 11.2781,E2 418.2114} C_DIS
LIN {X 115.0881,Y 68.672,Z 166,A 30.0762,B 11.1423,C 0.0858,E1 11.2818,E2 420.746} C_DIS
LIN {X 117.8602,Y 63.7986,Z 166,A 28.3144,B 11.1424,C 0.0756,E1 11.2841,E2 422.4336} C_DIS
LIN {X 120.6261,Y 58.3986,Z 166,A 25.933,B 11.1424,C 0.0768,E1 11.287,E2 424.7912} C_DIS
LIN {X 122.3828,Y 54.6173,Z 166,A 24.1026,B 11.1424,C 0.0827,E1 11.2891,E2 426.6287} C_DIS
LIN {X 123.7611,Y 51.4182,Z 166,A 22.609,B 11.1424,C 0.0868,E1 11.2908,E2 428.1239} C_DIS
LIN {X 125.4148,Y 47.2418,Z 166,A 20.6722,B 11.1423,C 0.0925,E1 11.2927,E2 430.0642} C_DIS
LIN {X 126.7159,Y 43.6321,Z 166,A 19.0603,B 11.1423,C 0.0962,E1 11.2942,E2 431.674} C_DIS
LIN {X 128.9057,Y 36.6646,Z 166,A 15.7263,B 11.1421,C 0.1105,E1 11.297,E2 435.0362} C_DIS
LIN {X 129.7809,Y 33.4332,Z 166,A 14.769,B 11.1421,C 0.1021,E1 11.2976,E2 435.9376} C_DIS
LIN {X 130.7665,Y 29.3433,Z 166,A 12.8844,B 11.1421,C 0.1095,E1 11.2988,E2 437.8342} C_DIS
LIN {X 131.491,Y 25.9106,Z 166,A 11.2453,B 11.1421,C 0.1174,E1 11.2997,E2 439.4916} C_DIS
LIN {X 132.2661,Y 21.5998,Z 166,A 9.5573,B 11.1421,C 0.1179,E1 11.3005,E2 441.159} C_DIS
LIN {X 132.7878,Y 18.1274,Z 166,A 7.9264,B 11.142,C 0.1257,E1 11.3012,E2 442.807} C_DIS
LIN {X 133.2425,Y 14.3915,Z 166,A 6.4867,B 11.142,C 0.1259,E1 11.3016,E2 444.2277} C_DIS
LIN {X 133.5686,Y 10.9642,Z 166,A 5.0667,B 11.142,C 0.1289,E1 11.302,E2 445.6429} C_DIS
Enddeposition()
END
